LIN {X 0,Y 312.474,Z 713.562,A -85,B 0,C 180,E1 -15779.659,E2 -15779.659} C_VEL
LIN {X 0,Y 312.526,Z 713.531,A -85,B 0,C 180,E1 -15783.69,E2 -15783.69} C_VEL
LIN {X 0,Y 312.516,Z 713.544,A -85,B 0,C 180,E1 -15787.388,E2 -15787.388} C_VEL
LIN {X 0,Y 312.441,Z 713.564,A -85,B 0,C 180,E1 -15790.719,E2 -15790.719} C_VEL
LIN {X 0,Y 312.452,Z 713.564,A -85,B 0,C 180,E1 -15794.212,E2 -15794.212} C_VEL
LIN {X 0,Y 312.461,Z 713.565,A -85,B 0,C 180,E1 -15797.926,E2 -15797.926} C_VEL
LIN {X 0,Y 312.482,Z 713.562,A -85,B 0,C 180,E1 -15801.925,E2 -15801.925} C_VEL
LIN {X 0,Y 312.497,Z 713.558,A -85,B 0,C 180,E1 -15802.312,E2 -15802.312} C_VEL
LIN {X 0,Y 312.585,Z 714.3,A -85,B 0,C 180,E1 -15802.882,E2 -15802.882} C_VEL
LIN {X 0,Y 312.799,Z 716.737,A -85,B 0,C 180,E1 -15803.505,E2 -15803.505} C_VEL
LIN {X 0,Y 313.144,Z 721.496,A -85,B 0,C 180,E1 -15804.133,E2 -15804.133} C_VEL
LIN {X 0,Y 313.458,Z 727.496,A -85,B 0,C 180,E1 -15804.555,E2 -15804.555} C_VEL
LIN {X 0,Y 313.606,Z 731.828,A -85,B 0,C 180,E1 -15804.761,E2 -15804.761} C_VEL
LIN {X 0,Y 313.578,Z 740.657,A -85,B 0,C 180,E1 -15805.058,E2 -15805.058} C_VEL
LIN {X 0,Y 312.273,Z 790.691,A -85,B 0,C 180,E1 -15806.517,E2 -15806.517} C_VEL
LIN {X 0,Y 311.933,Z 803.373,A -85,B 0,C 180,E1 -15807.082,E2 -15807.082} C_VEL
LIN {X 0,Y 311.545,Z 814.797,A -85,B 0,C 180,E1 -15807.795,E2 -15807.795} C_VEL
LIN {X 0,Y 311.035,Z 823.817,A -85,B 0,C 180,E1 -15808.498,E2 -15808.498} C_VEL
LIN {X 0,Y 310.379,Z 833.968,A -85,B 0,C 180,E1 -15809.476,E2 -15809.476} C_VEL
LIN {X 0,Y 309.692,Z 843.6,A -85,B 0,C 180,E1 -15810.61,E2 -15810.61} C_VEL
LIN {X 0,Y 308.984,Z 852.175,A -85,B 0,C 180,E1 -15811.813,E2 -15811.813} C_VEL
LIN {X 0,Y 308.32,Z 860.705,A -85,B 0,C 180,E1 -15813.244,E2 -15813.244} C_VEL
LIN {X 0,Y 307.678,Z 867.783,A -85,B 0,C 180,E1 -15814.641,E2 -15814.641} C_VEL
LIN {X 0,Y 307.055,Z 874.035,A -85,B 0,C 180,E1 -15816.084,E2 -15816.084} C_VEL
LIN {X 0,Y 306.572,Z 880.144,A -85,B 0,C 180,E1 -15817.774,E2 -15817.774} C_VEL
LIN {X 0,Y 306.255,Z 884.439,A -85,B 0,C 180,E1 -15819.163,E2 -15819.163} C_VEL
LIN {X 0,Y 305.896,Z 889.538,A -85,B 0,C 180,E1 -15821.237,E2 -15821.237} C_VEL
LIN {X 0,Y 305.687,Z 893.372,A -85,B 0,C 180,E1 -15823.298,E2 -15823.298} C_VEL
LIN {X 0,Y 305.662,Z 896.085,A -85,B 0,C 180,E1 -15825.349,E2 -15825.349} C_VEL
LIN {X 0,Y 305.728,Z 897.387,A -85,B 0,C 180,E1 -15826.71,E2 -15826.71} C_VEL
LIN {X 0,Y 305.909,Z 898.143,A -85,B 0,C 180,E1 -15828.067,E2 -15828.067} C_VEL
LIN {X 0,Y 306.419,Z 898.401,A -85,B 0,C 180,E1 -15830.495,E2 -15830.495} C_VEL
LIN {X 0,Y 306.824,Z 897.718,A -85,B 0,C 180,E1 -15832.1,E2 -15832.1} C_VEL
LIN {X 0,Y 307.906,Z 895.323,A -85,B 0,C 180,E1 -15834.761,E2 -15834.761} C_VEL
LIN {X 0,Y 308.867,Z 892.287,A -85,B 0,C 180,E1 -15836.739,E2 -15836.739} C_VEL
LIN {X 0,Y 309.999,Z 888.123,A -85,B 0,C 180,E1 -15838.701,E2 -15838.701} C_VEL
LIN {X 0,Y 311.371,Z 882.681,A -85,B 0,C 180,E1 -15840.646,E2 -15840.646} C_VEL
LIN {X 0,Y 312.733,Z 877.075,A -85,B 0,C 180,E1 -15842.254,E2 -15842.254} C_VEL
LIN {X 0,Y 314.123,Z 870.334,A -85,B 0,C 180,E1 -15843.848,E2 -15843.848} C_VEL
LIN {X 0,Y 315.423,Z 864,A -85,B 0,C 180,E1 -15845.113,E2 -15845.113} C_VEL
LIN {X 0,Y 317.072,Z 854.397,A -85,B 0,C 180,E1 -15846.682,E2 -15846.682} C_VEL
LIN {X 0,Y 318.271,Z 846.362,A -85,B 0,C 180,E1 -15847.773,E2 -15847.773} C_VEL
LIN {X 0,Y 319.492,Z 836.672,A -85,B 0,C 180,E1 -15848.858,E2 -15848.858} C_VEL
LIN {X 0,Y 320.502,Z 826.458,A -85,B 0,C 180,E1 -15849.784,E2 -15849.784} C_VEL
LIN {X 0,Y 321.27,Z 816.948,A -85,B 0,C 180,E1 -15850.477,E2 -15850.477} C_VEL
LIN {X 0,Y 321.877,Z 806.465,A -85,B 0,C 180,E1 -15851.069,E2 -15851.069} C_VEL
LIN {X 0,Y 322.31,Z 791.848,A -85,B 0,C 180,E1 -15851.674,E2 -15851.674} C_VEL
LIN {X 0,Y 324.232,Z 756.607,A -85,B 0,C 180,E1 -15852.839,E2 -15852.839} C_VEL
LIN {X 0,Y 324.778,Z 747.442,A -85,B 0,C 180,E1 -15853.145,E2 -15853.145} C_VEL
LIN {X 0,Y 319.601,Z 737.334,A -85,B 0,C 180,E1 -15854.411,E2 -15854.411} C_VEL
LIN {X 0,Y 314.132,Z 727.873,A -85,B 0,C 180,E1 -15855.834,E2 -15855.834} C_VEL
LIN {X 0,Y 310.936,Z 723.294,A -85,B 0,C 180,E1 -15856.678,E2 -15856.678} C_VEL
LIN {X 0,Y 308.894,Z 719.974,A -85,B 0,C 180,E1 -15857.287,E2 -15857.287} C_VEL
LIN {X 0,Y 306.255,Z 716.727,A -85,B 0,C 180,E1 -15858.04,E2 -15858.04} C_VEL
LIN {X 0,Y 305.63,Z 714.906,A -85,B 0,C 180,E1 -15858.397,E2 -15858.397} C_VEL
LIN {X 0,Y 305.556,Z 714.458,A -85,B 0,C 180,E1 -15858.784,E2 -15858.784} C_VEL
LIN {X 0,Y 305.494,Z 714.431,A -85,B 0,C 180,E1 -15863.039,E2 -15863.039} C_VEL
LIN {X 0,Y 305.485,Z 714.434,A -85,B 0,C 180,E1 -15866.199,E2 -15866.199} C_VEL
LIN {X 0,Y 305.47,Z 714.433,A -85,B 0,C 180,E1 -15869.038,E2 -15869.038} C_VEL
LIN {X 0,Y 305.444,Z 714.437,A -85,B 0,C 180,E1 -15871.952,E2 -15871.952} C_VEL
LIN {X 0,Y 305.469,Z 714.433,A -85,B 0,C 180,E1 -15875.112,E2 -15875.112} C_VEL
LIN {X 0,Y 305.474,Z 714.432,A -85,B 0,C 180,E1 -15878.532,E2 -15878.532} C_VEL
LIN {X 0,Y 305.462,Z 714.434,A -85,B 0,C 180,E1 -15882.585,E2 -15882.585} C_VEL
LIN {X 0,Y 305.432,Z 714.44,A -85,B 0,C 180,E1 -15886.344,E2 -15886.344} C_VEL
LIN {X 0,Y 305.465,Z 714.437,A -85,B 0,C 180,E1 -15889.891,E2 -15889.891} C_VEL
LIN {X 0,Y 305.548,Z 714.64,A -85,B 0,C 180,E1 -15891.024,E2 -15891.024} C_VEL
LIN {X 0,Y 308.834,Z 727.96,A -85,B 0,C 180,E1 -15894.5,E2 -15894.5} C_VEL
LIN {X 0,Y 312.064,Z 742.523,A -85,B 0,C 180,E1 -15898.044,E2 -15898.044} C_VEL
LIN {X 0,Y 312.777,Z 746.093,A -85,B 0,C 180,E1 -15898.88,E2 -15898.88} C_VEL
LIN {X 0,Y 312.679,Z 749.371,A -85,B 0,C 180,E1 -15899.479,E2 -15899.479} C_VEL
LIN {X 0,Y 316.155,Z 773.114,A -85,B 0,C 180,E1 -15901.211,E2 -15901.211} C_VEL
LIN {X 0,Y 318.854,Z 797.479,A -85,B 0,C 180,E1 -15902.693,E2 -15902.693} C_VEL
LIN {X 0,Y 319.866,Z 811.457,A -85,B 0,C 180,E1 -15903.412,E2 -15903.412} C_VEL
LIN {X 0,Y 320.681,Z 834.523,A -85,B 0,C 180,E1 -15904.458,E2 -15904.458} C_VEL
LIN {X 0,Y 318.329,Z 876.074,A -85,B 0,C 180,E1 -15905.805,E2 -15905.805} C_VEL
LIN {X 0,Y 317.232,Z 887.509,A -85,B 0,C 180,E1 -15906.323,E2 -15906.323} C_VEL
LIN {X 0,Y 315.932,Z 898.532,A -85,B 0,C 180,E1 -15907.001,E2 -15907.001} C_VEL
LIN {X 0,Y 314.124,Z 911.078,A -85,B 0,C 180,E1 -15907.989,E2 -15907.989} C_VEL
LIN {X 0,Y 312.112,Z 923.208,A -85,B 0,C 180,E1 -15909.226,E2 -15909.226} C_VEL
LIN {X 0,Y 310.105,Z 934.166,A -85,B 0,C 180,E1 -15910.641,E2 -15910.641} C_VEL
LIN {X 0,Y 308.519,Z 943.318,A -85,B 0,C 180,E1 -15912.088,E2 -15912.088} C_VEL
LIN {X 0,Y 307.446,Z 950.333,A -85,B 0,C 180,E1 -15913.395,E2 -15913.395} C_VEL
LIN {X 0,Y 306.228,Z 957.721,A -85,B 0,C 180,E1 -15915.001,E2 -15915.001} C_VEL
LIN {X 0,Y 305.272,Z 965.314,A -85,B 0,C 180,E1 -15917.027,E2 -15917.027} C_VEL
LIN {X 0,Y 304.626,Z 972.881,A -85,B 0,C 180,E1 -15919.362,E2 -15919.362} C_VEL
LIN {X 0,Y 304.487,Z 978.046,A -85,B 0,C 180,E1 -15921.369,E2 -15921.369} C_VEL
LIN {X 0,Y 304.547,Z 982.046,A -85,B 0,C 180,E1 -15923.372,E2 -15923.372} C_VEL
LIN {X 0,Y 304.686,Z 984.103,A -85,B 0,C 180,E1 -15924.704,E2 -15924.704} C_VEL
LIN {X 0,Y 304.883,Z 985.727,A -85,B 0,C 180,E1 -15926.033,E2 -15926.033} C_VEL
LIN {X 0,Y 304.952,Z 986.88,A -85,B 0,C 180,E1 -15927.356,E2 -15927.356} C_VEL
LIN {X 0,Y 305.065,Z 987.581,A -85,B 0,C 180,E1 -15928.678,E2 -15928.678} C_VEL
LIN {X 0,Y 305.169,Z 987.868,A -85,B 0,C 180,E1 -15929.998,E2 -15929.998} C_VEL
LIN {X 0,Y 305.046,Z 987.713,A -85,B 0,C 180,E1 -15931.318,E2 -15931.318} C_VEL
LIN {X 0,Y 304.924,Z 987.132,A -85,B 0,C 180,E1 -15932.64,E2 -15932.64} C_VEL
LIN {X 0,Y 304.873,Z 986.11,A -85,B 0,C 180,E1 -15933.964,E2 -15933.964} C_VEL
LIN {X 0,Y 304.544,Z 982.776,A -85,B 0,C 180,E1 -15936.624,E2 -15936.624} C_VEL
LIN {X 0,Y 304.4,Z 979.067,A -85,B 0,C 180,E1 -15938.629,E2 -15938.629} C_VEL
LIN {X 0,Y 304.57,Z 974.278,A -85,B 0,C 180,E1 -15940.636,E2 -15940.636} C_VEL
LIN {X 0,Y 305.237,Z 967.143,A -85,B 0,C 180,E1 -15942.971,E2 -15942.971} C_VEL
LIN {X 0,Y 306.243,Z 959.332,A -85,B 0,C 180,E1 -15944.992,E2 -15944.992} C_VEL
LIN {X 0,Y 307.609,Z 950.031,A -85,B 0,C 180,E1 -15946.934,E2 -15946.934} C_VEL
LIN {X 0,Y 309.193,Z 940.33,A -85,B 0,C 180,E1 -15948.553,E2 -15948.553} C_VEL
LIN {X 0,Y 310.906,Z 929.646,A -85,B 0,C 180,E1 -15949.99,E2 -15949.99} C_VEL
LIN {X 0,Y 312.682,Z 917.833,A -85,B 0,C 180,E1 -15951.247,E2 -15951.247} C_VEL
LIN {X 0,Y 314.307,Z 905.31,A -85,B 0,C 180,E1 -15952.253,E2 -15952.253} C_VEL
LIN {X 0,Y 315.703,Z 892.229,A -85,B 0,C 180,E1 -15953.012,E2 -15953.012} C_VEL
LIN {X 0,Y 316.491,Z 879.543,A -85,B 0,C 180,E1 -15953.514,E2 -15953.514} C_VEL
LIN {X 0,Y 317.678,Z 830.97,A -85,B 0,C 180,E1 -15954.672,E2 -15954.672} C_VEL
LIN {X 0,Y 314.724,Z 799.143,A -85,B 0,C 180,E1 -15955.761,E2 -15955.761} C_VEL
LIN {X 0,Y 311.458,Z 773.975,A -85,B 0,C 180,E1 -15956.747,E2 -15956.747} C_VEL
LIN {X 0,Y 310.704,Z 768.362,A -85,B 0,C 180,E1 -15957.031,E2 -15957.031} C_VEL
LIN {X 0,Y 313.403,Z 749.284,A -85,B 0,C 180,E1 -15961.046,E2 -15961.046} C_VEL
LIN {X 0,Y 313.001,Z 745.438,A -85,B 0,C 180,E1 -15961.962,E2 -15961.962} C_VEL
LIN {X 0,Y 310.448,Z 733.482,A -85,B 0,C 180,E1 -15965.026,E2 -15965.026} C_VEL
LIN {X 0,Y 307.708,Z 722.464,A -85,B 0,C 180,E1 -15968.071,E2 -15968.071} C_VEL
LIN {X 0,Y 305.475,Z 714.541,A -85,B 0,C 180,E1 -15970.484,E2 -15970.484} C_VEL
LIN {X 0,Y 305.435,Z 714.433,A -85,B 0,C 180,E1 -15973.65,E2 -15973.65} C_VEL
LIN {X 0,Y 305.469,Z 714.432,A -85,B 0,C 180,E1 -15977.408,E2 -15977.408} C_VEL
LIN {X 0,Y 305.486,Z 714.43,A -85,B 0,C 180,E1 -15981.599,E2 -15981.599} C_VEL
LIN {X 0,Y 305.453,Z 714.418,A -85,B 0,C 180,E1 -15984.886,E2 -15984.886} C_VEL
LIN {X 0,Y 305.442,Z 714.435,A -85,B 0,C 180,E1 -15988.354,E2 -15988.354} C_VEL
LIN {X 0,Y 305.51,Z 714.428,A -85,B 0,C 180,E1 -15991.113,E2 -15991.113} C_VEL
LIN {X 0,Y 305.561,Z 714.42,A -85,B 0,C 180,E1 -15994.087,E2 -15994.087} C_VEL
LIN {X 0,Y 305.489,Z 714.424,A -85,B 0,C 180,E1 -15998.402,E2 -15998.402} C_VEL
LIN {X 0,Y 305.579,Z 714.421,A -85,B 0,C 180,E1 -16001.217,E2 -16001.217} C_VEL
LIN {X 0,Y 305.638,Z 714.414,A -85,B 0,C 180,E1 -16005.349,E2 -16005.349} C_VEL
LIN {X 0,Y 305.624,Z 714.415,A -85,B 0,C 180,E1 -16009.399,E2 -16009.399} C_VEL
LIN {X 0,Y 305.784,Z 714.387,A -85,B 0,C 180,E1 -16012.074,E2 -16012.074} C_VEL
LIN {X 0,Y 305.676,Z 714.402,A -85,B 0,C 180,E1 -16014.723,E2 -16014.723} C_VEL
LIN {X 0,Y 305.946,Z 714.372,A -85,B 0,C 180,E1 -16018.684,E2 -16018.684} C_VEL
LIN {X 0,Y 305.945,Z 714.371,A -85,B 0,C 180,E1 -16021.317,E2 -16021.317} C_VEL
LIN {X 0,Y 305.84,Z 714.39,A -85,B 0,C 180,E1 -16026.598,E2 -16026.598} C_VEL
LIN {X 0,Y 305.724,Z 714.397,A -85,B 0,C 180,E1 -16029.26,E2 -16029.26} C_VEL
LIN {X 0,Y 305.578,Z 714.418,A -85,B 0,C 180,E1 -16033.297,E2 -16033.297} C_VEL
LIN {X 0,Y 305.583,Z 714.412,A -85,B 0,C 180,E1 -16036.021,E2 -16036.021} C_VEL
LIN {X 0,Y 305.549,Z 714.42,A -85,B 0,C 180,E1 -16039.437,E2 -16039.437} C_VEL
LIN {X 0,Y 305.476,Z 714.414,A -85,B 0,C 180,E1 -16043.041,E2 -16043.041} C_VEL
LIN {X 0,Y 305.543,Z 714.428,A -85,B 0,C 180,E1 -16046.23,E2 -16046.23} C_VEL
LIN {X 0,Y 305.478,Z 714.419,A -85,B 0,C 180,E1 -16049.049,E2 -16049.049} C_VEL
LIN {X 0,Y 305.433,Z 714.431,A -85,B 0,C 180,E1 -16051.954,E2 -16051.954} C_VEL
LIN {X 0,Y 305.454,Z 714.432,A -85,B 0,C 180,E1 -16055.115,E2 -16055.115} C_VEL
LIN {X 0,Y 305.527,Z 714.61,A -85,B 0,C 180,E1 -16057.872,E2 -16057.872} C_VEL
LIN {X 0,Y 305.73,Z 715.512,A -85,B 0,C 180,E1 -16058.103,E2 -16058.103} C_VEL
LIN {X 0,Y 315.424,Z 734.481,A -85,B 0,C 180,E1 -16059.68,E2 -16059.68} C_VEL
LIN {X 0,Y 319.798,Z 744.244,A -85,B 0,C 180,E1 -16060.363,E2 -16060.363} C_VEL
LIN {X 0,Y 318.757,Z 791.246,A -85,B 0,C 180,E1 -16061.487,E2 -16061.487} C_VEL
LIN {X 0,Y 318.629,Z 805.311,A -85,B 0,C 180,E1 -16061.953,E2 -16061.953} C_VEL
LIN {X 0,Y 318.217,Z 817.903,A -85,B 0,C 180,E1 -16062.635,E2 -16062.635} C_VEL
LIN {X 0,Y 317.446,Z 829.918,A -85,B 0,C 180,E1 -16063.529,E2 -16063.529} C_VEL
LIN {X 0,Y 316.275,Z 841.723,A -85,B 0,C 180,E1 -16064.68,E2 -16064.68} C_VEL
LIN {X 0,Y 315.059,Z 851.984,A -85,B 0,C 180,E1 -16065.965,E2 -16065.965} C_VEL
LIN {X 0,Y 313.601,Z 862.112,A -85,B 0,C 180,E1 -16067.539,E2 -16067.539} C_VEL
LIN {X 0,Y 312.162,Z 870.912,A -85,B 0,C 180,E1 -16069.242,E2 -16069.242} C_VEL
LIN {X 0,Y 310.744,Z 878.712,A -85,B 0,C 180,E1 -16071.129,E2 -16071.129} C_VEL
LIN {X 0,Y 309.477,Z 885.377,A -85,B 0,C 180,E1 -16073.155,E2 -16073.155} C_VEL
LIN {X 0,Y 308.311,Z 890.805,A -85,B 0,C 180,E1 -16075.261,E2 -16075.261} C_VEL
LIN {X 0,Y 307.625,Z 893.802,A -85,B 0,C 180,E1 -16076.752,E2 -16076.752} C_VEL
LIN {X 0,Y 307.12,Z 896.217,A -85,B 0,C 180,E1 -16078.245,E2 -16078.245} C_VEL
LIN {X 0,Y 306.516,Z 898.862,A -85,B 0,C 180,E1 -16080.61,E2 -16080.61} C_VEL
LIN {X 0,Y 306.113,Z 900.115,A -85,B 0,C 180,E1 -16082.668,E2 -16082.668} C_VEL
LIN {X 0,Y 305.972,Z 900.399,A -85,B 0,C 180,E1 -16084.127,E2 -16084.127} C_VEL
LIN {X 0,Y 305.894,Z 900.247,A -85,B 0,C 180,E1 -16085.574,E2 -16085.574} C_VEL
LIN {X 0,Y 305.928,Z 899.592,A -85,B 0,C 180,E1 -16087.014,E2 -16087.014} C_VEL
LIN {X 0,Y 306.068,Z 898.48,A -85,B 0,C 180,E1 -16088.447,E2 -16088.447} C_VEL
LIN {X 0,Y 306.371,Z 896.552,A -85,B 0,C 180,E1 -16090.141,E2 -16090.141} C_VEL
LIN {X 0,Y 307.026,Z 892.313,A -85,B 0,C 180,E1 -16092.69,E2 -16092.69} C_VEL
LIN {X 0,Y 307.806,Z 887.5,A -85,B 0,C 180,E1 -16094.779,E2 -16094.779} C_VEL
LIN {X 0,Y 308.726,Z 881.356,A -85,B 0,C 180,E1 -16096.844,E2 -16096.844} C_VEL
LIN {X 0,Y 309.865,Z 873.672,A -85,B 0,C 180,E1 -16098.887,E2 -16098.887} C_VEL
LIN {X 0,Y 310.965,Z 865.834,A -85,B 0,C 180,E1 -16100.571,E2 -16100.571} C_VEL
LIN {X 0,Y 312.203,Z 856.299,A -85,B 0,C 180,E1 -16102.24,E2 -16102.24} C_VEL
LIN {X 0,Y 313.404,Z 845.67,A -85,B 0,C 180,E1 -16103.726,E2 -16103.726} C_VEL
LIN {X 0,Y 314.523,Z 833.894,A -85,B 0,C 180,E1 -16105.035,E2 -16105.035} C_VEL
LIN {X 0,Y 315.393,Z 821.458,A -85,B 0,C 180,E1 -16106.089,E2 -16106.089} C_VEL
LIN {X 0,Y 315.943,Z 808.598,A -85,B 0,C 180,E1 -16106.894,E2 -16106.894} C_VEL
LIN {X 0,Y 316.171,Z 796.443,A -85,B 0,C 180,E1 -16107.414,E2 -16107.414} C_VEL
LIN {X 0,Y 316.968,Z 746.283,A -85,B 0,C 180,E1 -16108.625,E2 -16108.625} C_VEL
LIN {X 0,Y 317.049,Z 741.291,A -85,B 0,C 180,E1 -16108.743,E2 -16108.743} C_VEL
LIN {X 0,Y 309.365,Z 722.642,A -85,B 0,C 180,E1 -16109.816,E2 -16109.816} C_VEL
LIN {X 0,Y 306.062,Z 715.169,A -85,B 0,C 180,E1 -16110.331,E2 -16110.331} C_VEL
LIN {X 0,Y 305.923,Z 714.461,A -85,B 0,C 180,E1 -16110.578,E2 -16110.578} C_VEL
LIN {X 0,Y 305.85,Z 714.387,A -85,B 0,C 180,E1 -16112.636,E2 -16112.636} C_VEL
LIN {X 0,Y 305.788,Z 714.391,A -85,B 0,C 180,E1 -16116.601,E2 -16116.601} C_VEL
LIN {X 0,Y 305.698,Z 714.406,A -85,B 0,C 180,E1 -16119.263,E2 -16119.263} C_VEL
LIN {X 0,Y 305.589,Z 714.417,A -85,B 0,C 180,E1 -16123.298,E2 -16123.298} C_VEL
LIN {X 0,Y 305.554,Z 714.418,A -85,B 0,C 180,E1 -16126.024,E2 -16126.024} C_VEL
LIN {X 0,Y 305.485,Z 714.414,A -85,B 0,C 180,E1 -16130.189,E2 -16130.189} C_VEL
LIN {X 0,Y 305.461,Z 714.431,A -85,B 0,C 180,E1 -16134.467,E2 -16134.467} C_VEL
LIN {X 0,Y 305.447,Z 714.418,A -85,B 0,C 180,E1 -16137.401,E2 -16137.401} C_VEL
LIN {X 0,Y 305.421,Z 714.439,A -85,B 0,C 180,E1 -16140.416,E2 -16140.416} C_VEL
LIN {X 0,Y 305.471,Z 714.406,A -85,B 0,C 180,E1 -16144.079,E2 -16144.079} C_VEL
LIN {X 0,Y 305.458,Z 714.418,A -85,B 0,C 180,E1 -16146.744,E2 -16146.744} C_VEL
LIN {X 0,Y 305.412,Z 714.439,A -85,B 0,C 180,E1 -16150.59,E2 -16150.59} C_VEL
LIN {X 0,Y 305.402,Z 714.442,A -85,B 0,C 180,E1 -16154.489,E2 -16154.489} C_VEL
LIN {X 0,Y 305.418,Z 714.441,A -85,B 0,C 180,E1 -16158.139,E2 -16158.139} C_VEL
LIN {X 0,Y 305.444,Z 714.434,A -85,B 0,C 180,E1 -16162.318,E2 -16162.318} C_VEL
LIN {X 0,Y 305.515,Z 714.584,A -85,B 0,C 180,E1 -16163.626,E2 -16163.626} C_VEL
LIN {X 0,Y 305.74,Z 715.565,A -85,B 0,C 180,E1 -16163.847,E2 -16163.847} C_VEL
LIN {X 0,Y 313.568,Z 737.666,A -85,B 0,C 180,E1 -16164.965,E2 -16164.965} C_VEL
LIN {X 0,Y 313.578,Z 740.657,A -85,B 0,C 180,E1 -16165.058,E2 -16165.058} C_VEL
LIN {X 0,Y 312.734,Z 746.454,A -85,B 0,C 180,E1 -16165.195,E2 -16165.195} C_VEL
LIN {X 0,Y 306.578,Z 765.245,A -85,B 0,C 180,E1 -16165.463,E2 -16165.463} C_VEL
LIN {X 0,Y 305.777,Z 771.044,A -85,B 0,C 180,E1 -16165.605,E2 -16165.605} C_VEL
LIN {X 0,Y 305.326,Z 794.538,A -85,B 0,C 180,E1 -16166.36,E2 -16166.36} C_VEL
LIN {X 0,Y 305.001,Z 805.646,A -85,B 0,C 180,E1 -16166.894,E2 -16166.894} C_VEL
LIN {X 0,Y 304.593,Z 815.918,A -85,B 0,C 180,E1 -16167.557,E2 -16167.557} C_VEL
LIN {X 0,Y 304.024,Z 825.634,A -85,B 0,C 180,E1 -16168.343,E2 -16168.343} C_VEL
LIN {X 0,Y 303.35,Z 835.762,A -85,B 0,C 180,E1 -16169.356,E2 -16169.356} C_VEL
LIN {X 0,Y 302.706,Z 844.701,A -85,B 0,C 180,E1 -16170.438,E2 -16170.438} C_VEL
LIN {X 0,Y 301.987,Z 853.411,A -85,B 0,C 180,E1 -16171.694,E2 -16171.694} C_VEL
LIN {X 0,Y 301.387,Z 860.846,A -85,B 0,C 180,E1 -16172.953,E2 -16172.953} C_VEL
LIN {X 0,Y 300.712,Z 868.066,A -85,B 0,C 180,E1 -16174.382,E2 -16174.382} C_VEL
LIN {X 0,Y 300.009,Z 875.015,A -85,B 0,C 180,E1 -16176.014,E2 -16176.014} C_VEL
LIN {X 0,Y 299.496,Z 881.754,A -85,B 0,C 180,E1 -16177.947,E2 -16177.947} C_VEL
LIN {X 0,Y 299.161,Z 885.968,A -85,B 0,C 180,E1 -16179.366,E2 -16179.366} C_VEL
LIN {X 0,Y 298.805,Z 890.961,A -85,B 0,C 180,E1 -16181.486,E2 -16181.486} C_VEL
LIN {X 0,Y 298.635,Z 894.723,A -85,B 0,C 180,E1 -16183.596,E2 -16183.596} C_VEL
LIN {X 0,Y 298.642,Z 896.698,A -85,B 0,C 180,E1 -16184.997,E2 -16184.997} C_VEL
LIN {X 0,Y 298.85,Z 899.05,A -85,B 0,C 180,E1 -16187.781,E2 -16187.781} C_VEL
LIN {X 0,Y 299.107,Z 899.551,A -85,B 0,C 180,E1 -16189.165,E2 -16189.165} C_VEL
LIN {X 0,Y 299.431,Z 899.584,A -85,B 0,C 180,E1 -16190.543,E2 -16190.543} C_VEL
LIN {X 0,Y 300.297,Z 898.379,A -85,B 0,C 180,E1 -16193.28,E2 -16193.28} C_VEL
LIN {X 0,Y 300.883,Z 897.05,A -85,B 0,C 180,E1 -16194.639,E2 -16194.639} C_VEL
LIN {X 0,Y 302.263,Z 893.151,A -85,B 0,C 180,E1 -16197.334,E2 -16197.334} C_VEL
LIN {X 0,Y 303.496,Z 888.881,A -85,B 0,C 180,E1 -16199.336,E2 -16199.336} C_VEL
LIN {X 0,Y 304.999,Z 883.346,A -85,B 0,C 180,E1 -16201.32,E2 -16201.32} C_VEL
LIN {X 0,Y 306.479,Z 877.671,A -85,B 0,C 180,E1 -16202.957,E2 -16202.957} C_VEL
LIN {X 0,Y 307.681,Z 872.391,A -85,B 0,C 180,E1 -16204.257,E2 -16204.257} C_VEL
LIN {X 0,Y 309.386,Z 864.367,A -85,B 0,C 180,E1 -16205.867,E2 -16205.867} C_VEL
LIN {X 0,Y 310.799,Z 856.743,A -85,B 0,C 180,E1 -16207.144,E2 -16207.144} C_VEL
LIN {X 0,Y 312.264,Z 847.644,A -85,B 0,C 180,E1 -16208.412,E2 -16208.412} C_VEL
LIN {X 0,Y 313.528,Z 838.356,A -85,B 0,C 180,E1 -16209.487,E2 -16209.487} C_VEL
LIN {X 0,Y 314.524,Z 829.875,A -85,B 0,C 180,E1 -16210.297,E2 -16210.297} C_VEL
LIN {X 0,Y 315.362,Z 819.879,A -85,B 0,C 180,E1 -16211.082,E2 -16211.082} C_VEL
LIN {X 0,Y 316.103,Z 808.632,A -85,B 0,C 180,E1 -16211.746,E2 -16211.746} C_VEL
LIN {X 0,Y 316.552,Z 795.014,A -85,B 0,C 180,E1 -16212.339,E2 -16212.339} C_VEL
LIN {X 0,Y 318.225,Z 765.799,A -85,B 0,C 180,E1 -16213.349,E2 -16213.349} C_VEL
LIN {X 0,Y 319.277,Z 750.021,A -85,B 0,C 180,E1 -16213.886,E2 -16213.886} C_VEL
LIN {X 0,Y 313.25,Z 738.49,A -85,B 0,C 180,E1 -16215.462,E2 -16215.462} C_VEL
LIN {X 0,Y 308.903,Z 731.443,A -85,B 0,C 180,E1 -16216.657,E2 -16216.657} C_VEL
LIN {X 0,Y 306.662,Z 728.003,A -85,B 0,C 180,E1 -16217.323,E2 -16217.323} C_VEL
LIN {X 0,Y 304.411,Z 724.587,A -85,B 0,C 180,E1 -16218.007,E2 -16218.007} C_VEL
LIN {X 0,Y 302.286,Z 721.473,A -85,B 0,C 180,E1 -16218.691,E2 -16218.691} C_VEL
LIN {X 0,Y 301.699,Z 720.414,A -85,B 0,C 180,E1 -16218.899,E2 -16218.899} C_VEL
LIN {X 0,Y 299.389,Z 717.967,A -85,B 0,C 180,E1 -16219.633,E2 -16219.633} C_VEL
LIN {X 0,Y 298.573,Z 715.892,A -85,B 0,C 180,E1 -16220.072,E2 -16220.072} C_VEL
LIN {X 0,Y 298.441,Z 715.323,A -85,B 0,C 180,E1 -16220.685,E2 -16220.685} C_VEL
LIN {X 0,Y 298.457,Z 715.306,A -85,B 0,C 180,E1 -16225.078,E2 -16225.078} C_VEL
LIN {X 0,Y 298.418,Z 715.314,A -85,B 0,C 180,E1 -16229.377,E2 -16229.377} C_VEL
LIN {X 0,Y 298.4,Z 715.313,A -85,B 0,C 180,E1 -16232.8,E2 -16232.8} C_VEL
LIN {X 0,Y 298.458,Z 715.305,A -85,B 0,C 180,E1 -16236.808,E2 -16236.808} C_VEL
LIN {X 0,Y 298.416,Z 715.312,A -85,B 0,C 180,E1 -16239.485,E2 -16239.485} C_VEL
LIN {X 0,Y 298.405,Z 715.312,A -85,B 0,C 180,E1 -16243.102,E2 -16243.102} C_VEL
LIN {X 0,Y 298.409,Z 715.312,A -85,B 0,C 180,E1 -16246.92,E2 -16246.92} C_VEL
LIN {X 0,Y 298.465,Z 715.403,A -85,B 0,C 180,E1 -16250.411,E2 -16250.411} C_VEL
LIN {X 0,Y 299.21,Z 718.35,A -85,B 0,C 180,E1 -16251.304,E2 -16251.304} C_VEL
LIN {X 0,Y 302.683,Z 732.696,A -85,B 0,C 180,E1 -16255.07,E2 -16255.07} C_VEL
LIN {X 0,Y 304.493,Z 740.8,A -85,B 0,C 180,E1 -16257.065,E2 -16257.065} C_VEL
LIN {X 0,Y 306.204,Z 747.221,A -85,B 0,C 180,E1 -16258.135,E2 -16258.135} C_VEL
LIN {X 0,Y 307.688,Z 752.126,A -85,B 0,C 180,E1 -16258.693,E2 -16258.693} C_VEL
LIN {X 0,Y 310.905,Z 775.277,A -85,B 0,C 180,E1 -16260.438,E2 -16260.438} C_VEL
LIN {X 0,Y 313.325,Z 798.973,A -85,B 0,C 180,E1 -16261.934,E2 -16261.934} C_VEL
LIN {X 0,Y 314.23,Z 813.346,A -85,B 0,C 180,E1 -16262.706,E2 -16262.706} C_VEL
LIN {X 0,Y 314.908,Z 835.446,A -85,B 0,C 180,E1 -16263.729,E2 -16263.729} C_VEL
LIN {X 0,Y 312.474,Z 874.755,A -85,B 0,C 180,E1 -16265.055,E2 -16265.055} C_VEL
LIN {X 0,Y 311.232,Z 886.765,A -85,B 0,C 180,E1 -16265.616,E2 -16265.616} C_VEL
LIN {X 0,Y 309.486,Z 900.437,A -85,B 0,C 180,E1 -16266.494,E2 -16266.494} C_VEL
LIN {X 0,Y 307.327,Z 913.607,A -85,B 0,C 180,E1 -16267.653,E2 -16267.653} C_VEL
LIN {X 0,Y 305.506,Z 923.608,A -85,B 0,C 180,E1 -16268.755,E2 -16268.755} C_VEL
LIN {X 0,Y 303.676,Z 933.179,A -85,B 0,C 180,E1 -16270.038,E2 -16270.038} C_VEL
LIN {X 0,Y 302.14,Z 941.379,A -85,B 0,C 180,E1 -16271.345,E2 -16271.345} C_VEL
LIN {X 0,Y 300.816,Z 948.49,A -85,B 0,C 180,E1 -16272.668,E2 -16272.668} C_VEL
LIN {X 0,Y 299.392,Z 956.315,A -85,B 0,C 180,E1 -16274.411,E2 -16274.411} C_VEL
LIN {X 0,Y 298.416,Z 963.57,A -85,B 0,C 180,E1 -16276.376,E2 -16276.376} C_VEL
LIN {X 0,Y 297.742,Z 969.781,A -85,B 0,C 180,E1 -16278.424,E2 -16278.424} C_VEL
LIN {X 0,Y 297.451,Z 975.316,A -85,B 0,C 180,E1 -16280.478,E2 -16280.478} C_VEL
LIN {X 0,Y 297.453,Z 980.432,A -85,B 0,C 180,E1 -16282.907,E2 -16282.907} C_VEL
LIN {X 0,Y 297.617,Z 983.026,A -85,B 0,C 180,E1 -16284.578,E2 -16284.578} C_VEL
LIN {X 0,Y 297.836,Z 984.665,A -85,B 0,C 180,E1 -16285.939,E2 -16285.939} C_VEL
LIN {X 0,Y 297.908,Z 985.84,A -85,B 0,C 180,E1 -16287.294,E2 -16287.294} C_VEL
LIN {X 0,Y 298.028,Z 986.554,A -85,B 0,C 180,E1 -16288.647,E2 -16288.647} C_VEL
LIN {X 0,Y 298.139,Z 986.852,A -85,B 0,C 180,E1 -16289.998,E2 -16289.998} C_VEL
LIN {X 0,Y 298.007,Z 986.704,A -85,B 0,C 180,E1 -16291.349,E2 -16291.349} C_VEL
LIN {X 0,Y 297.877,Z 986.139,A -85,B 0,C 180,E1 -16292.703,E2 -16292.703} C_VEL
LIN {X 0,Y 297.804,Z 985.124,A -85,B 0,C 180,E1 -16294.058,E2 -16294.058} C_VEL
LIN {X 0,Y 297.567,Z 983.666,A -85,B 0,C 180,E1 -16295.419,E2 -16295.419} C_VEL
LIN {X 0,Y 297.428,Z 981.381,A -85,B 0,C 180,E1 -16297.055,E2 -16297.055} C_VEL
LIN {X 0,Y 297.344,Z 976.633,A -85,B 0,C 180,E1 -16299.521,E2 -16299.521} C_VEL
LIN {X 0,Y 297.679,Z 971.482,A -85,B 0,C 180,E1 -16301.575,E2 -16301.575} C_VEL
LIN {X 0,Y 298.347,Z 965.075,A -85,B 0,C 180,E1 -16303.623,E2 -16303.623} C_VEL
LIN {X 0,Y 299.226,Z 958.883,A -85,B 0,C 180,E1 -16305.253,E2 -16305.253} C_VEL
LIN {X 0,Y 300.762,Z 949.241,A -85,B 0,C 180,E1 -16307.331,E2 -16307.331} C_VEL
LIN {X 0,Y 302.455,Z 939.616,A -85,B 0,C 180,E1 -16308.982,E2 -16308.982} C_VEL
LIN {X 0,Y 304.246,Z 929.001,A -85,B 0,C 180,E1 -16310.447,E2 -16310.447} C_VEL
LIN {X 0,Y 305.791,Z 918.876,A -85,B 0,C 180,E1 -16311.573,E2 -16311.573} C_VEL
LIN {X 0,Y 307.475,Z 907.101,A -85,B 0,C 180,E1 -16312.597,E2 -16312.597} C_VEL
LIN {X 0,Y 308.941,Z 894.403,A -85,B 0,C 180,E1 -16313.413,E2 -16313.413} C_VEL
LIN {X 0,Y 309.945,Z 881.094,A -85,B 0,C 180,E1 -16313.997,E2 -16313.997} C_VEL
LIN {X 0,Y 310.793,Z 855.297,A -85,B 0,C 180,E1 -16314.653,E2 -16314.653} C_VEL
LIN {X 0,Y 311.281,Z 831.143,A -85,B 0,C 180,E1 -16315.242,E2 -16315.242} C_VEL
LIN {X 0,Y 308.408,Z 799.908,A -85,B 0,C 180,E1 -16316.35,E2 -16316.35} C_VEL
LIN {X 0,Y 305.525,Z 777.341,A -85,B 0,C 180,E1 -16317.255,E2 -16317.255} C_VEL
LIN {X 0,Y 304.078,Z 767.429,A -85,B 0,C 180,E1 -16317.719,E2 -16317.719} C_VEL
LIN {X 0,Y 306.633,Z 750.18,A -85,B 0,C 180,E1 -16321.425,E2 -16321.425} C_VEL
LIN {X 0,Y 304.61,Z 739.442,A -85,B 0,C 180,E1 -16324.182,E2 -16324.182} C_VEL
LIN {X 0,Y 301.678,Z 727.061,A -85,B 0,C 180,E1 -16327.62,E2 -16327.62} C_VEL
LIN {X 0,Y 298.837,Z 717.039,A -85,B 0,C 180,E1 -16330.672,E2 -16330.672} C_VEL
LIN {X 0,Y 298.398,Z 715.405,A -85,B 0,C 180,E1 -16331.256,E2 -16331.256} C_VEL
LIN {X 0,Y 298.38,Z 715.315,A -85,B 0,C 180,E1 -16335.04,E2 -16335.04} C_VEL
LIN {X 0,Y 298.404,Z 715.31,A -85,B 0,C 180,E1 -16338.742,E2 -16338.742} C_VEL
LIN {X 0,Y 298.422,Z 715.313,A -85,B 0,C 180,E1 -16342.243,E2 -16342.243} C_VEL
LIN {X 0,Y 298.398,Z 715.301,A -85,B 0,C 180,E1 -16345.58,E2 -16345.58} C_VEL
LIN {X 0,Y 298.385,Z 715.313,A -85,B 0,C 180,E1 -16348.79,E2 -16348.79} C_VEL
LIN {X 0,Y 298.459,Z 715.303,A -85,B 0,C 180,E1 -16351.904,E2 -16351.904} C_VEL
LIN {X 0,Y 298.475,Z 715.3,A -85,B 0,C 180,E1 -16354.923,E2 -16354.923} C_VEL
LIN {X 0,Y 298.439,Z 715.303,A -85,B 0,C 180,E1 -16359.315,E2 -16359.315} C_VEL
LIN {X 0,Y 298.526,Z 715.29,A -85,B 0,C 180,E1 -16362.179,E2 -16362.179} C_VEL
LIN {X 0,Y 298.582,Z 715.291,A -85,B 0,C 180,E1 -16364.994,E2 -16364.994} C_VEL
LIN {X 0,Y 298.58,Z 715.292,A -85,B 0,C 180,E1 -16369.146,E2 -16369.146} C_VEL
LIN {X 0,Y 298.729,Z 715.264,A -85,B 0,C 180,E1 -16371.885,E2 -16371.885} C_VEL
LIN {X 0,Y 298.646,Z 715.279,A -85,B 0,C 180,E1 -16374.599,E2 -16374.599} C_VEL
LIN {X 0,Y 298.912,Z 715.248,A -85,B 0,C 180,E1 -16378.653,E2 -16378.653} C_VEL
LIN {X 0,Y 298.912,Z 715.247,A -85,B 0,C 180,E1 -16381.347,E2 -16381.347} C_VEL
LIN {X 0,Y 298.785,Z 715.268,A -85,B 0,C 180,E1 -16386.754,E2 -16386.754} C_VEL
LIN {X 0,Y 298.669,Z 715.277,A -85,B 0,C 180,E1 -16389.481,E2 -16389.481} C_VEL
LIN {X 0,Y 298.541,Z 715.297,A -85,B 0,C 180,E1 -16393.616,E2 -16393.616} C_VEL
LIN {X 0,Y 298.538,Z 715.291,A -85,B 0,C 180,E1 -16396.41,E2 -16396.41} C_VEL
LIN {X 0,Y 298.487,Z 715.3,A -85,B 0,C 180,E1 -16399.648,E2 -16399.648} C_VEL
LIN {X 0,Y 298.418,Z 715.291,A -85,B 0,C 180,E1 -16403.601,E2 -16403.601} C_VEL
LIN {X 0,Y 298.481,Z 715.308,A -85,B 0,C 180,E1 -16406.576,E2 -16406.576} C_VEL
LIN {X 0,Y 298.407,Z 715.305,A -85,B 0,C 180,E1 -16409.643,E2 -16409.643} C_VEL
LIN {X 0,Y 298.386,Z 715.305,A -85,B 0,C 180,E1 -16412.802,E2 -16412.802} C_VEL
LIN {X 0,Y 298.492,Z 715.476,A -85,B 0,C 180,E1 -16417.072,E2 -16417.072} C_VEL
LIN {X 0,Y 298.761,Z 716.615,A -85,B 0,C 180,E1 -16417.343,E2 -16417.343} C_VEL
LIN {X 0,Y 307.419,Z 733.091,A -85,B 0,C 180,E1 -16418.805,E2 -16418.805} C_VEL
LIN {X 0,Y 313.512,Z 746.196,A -85,B 0,C 180,E1 -16419.801,E2 -16419.801} C_VEL
LIN {X 0,Y 312.432,Z 792.282,A -85,B 0,C 180,E1 -16420.926,E2 -16420.926} C_VEL
LIN {X 0,Y 312.298,Z 805.781,A -85,B 0,C 180,E1 -16421.375,E2 -16421.375} C_VEL
LIN {X 0,Y 311.939,Z 817.079,A -85,B 0,C 180,E1 -16421.974,E2 -16421.974} C_VEL
LIN {X 0,Y 311.204,Z 828.851,A -85,B 0,C 180,E1 -16422.83,E2 -16422.83} C_VEL
LIN {X 0,Y 310.08,Z 840.427,A -85,B 0,C 180,E1 -16423.928,E2 -16423.928} C_VEL
LIN {X 0,Y 308.903,Z 850.544,A -85,B 0,C 180,E1 -16425.15,E2 -16425.15} C_VEL
LIN {X 0,Y 307.402,Z 860.839,A -85,B 0,C 180,E1 -16426.699,E2 -16426.699} C_VEL
LIN {X 0,Y 305.993,Z 869.13,A -85,B 0,C 180,E1 -16428.239,E2 -16428.239} C_VEL
LIN {X 0,Y 304.45,Z 877.518,A -85,B 0,C 180,E1 -16430.167,E2 -16430.167} C_VEL
LIN {X 0,Y 303.199,Z 883.949,A -85,B 0,C 180,E1 -16432.009,E2 -16432.009} C_VEL
LIN {X 0,Y 302.196,Z 888.572,A -85,B 0,C 180,E1 -16433.63,E2 -16433.63} C_VEL
LIN {X 0,Y 300.966,Z 893.743,A -85,B 0,C 180,E1 -16435.917,E2 -16435.917} C_VEL
LIN {X 0,Y 300.117,Z 897.475,A -85,B 0,C 180,E1 -16438.207,E2 -16438.207} C_VEL
LIN {X 0,Y 299.546,Z 899.9,A -85,B 0,C 180,E1 -16440.484,E2 -16440.484} C_VEL
LIN {X 0,Y 299.201,Z 900.872,A -85,B 0,C 180,E1 -16441.982,E2 -16441.982} C_VEL
LIN {X 0,Y 299.027,Z 901.379,A -85,B 0,C 180,E1 -16443.48,E2 -16443.48} C_VEL
LIN {X 0,Y 298.897,Z 901.366,A -85,B 0,C 180,E1 -16444.963,E2 -16444.963} C_VEL
LIN {X 0,Y 298.884,Z 900.884,A -85,B 0,C 180,E1 -16446.5,E2 -16446.5} C_VEL
LIN {X 0,Y 298.997,Z 899.99,A -85,B 0,C 180,E1 -16447.911,E2 -16447.911} C_VEL
LIN {X 0,Y 299.289,Z 897.936,A -85,B 0,C 180,E1 -16449.935,E2 -16449.935} C_VEL
LIN {X 0,Y 299.882,Z 894.355,A -85,B 0,C 180,E1 -16452.264,E2 -16452.264} C_VEL
LIN {X 0,Y 300.601,Z 889.848,A -85,B 0,C 180,E1 -16454.405,E2 -16454.405} C_VEL
LIN {X 0,Y 301.542,Z 884.065,A -85,B 0,C 180,E1 -16456.524,E2 -16456.524} C_VEL
LIN {X 0,Y 302.677,Z 876.837,A -85,B 0,C 180,E1 -16458.619,E2 -16458.619} C_VEL
LIN {X 0,Y 304.003,Z 867.749,A -85,B 0,C 180,E1 -16460.689,E2 -16460.689} C_VEL
LIN {X 0,Y 305.282,Z 858.472,A -85,B 0,C 180,E1 -16462.386,E2 -16462.386} C_VEL
LIN {X 0,Y 306.541,Z 848.084,A -85,B 0,C 180,E1 -16463.915,E2 -16463.915} C_VEL
LIN {X 0,Y 307.681,Z 836.632,A -85,B 0,C 180,E1 -16465.252,E2 -16465.252} C_VEL
LIN {X 0,Y 308.644,Z 824.793,A -85,B 0,C 180,E1 -16466.33,E2 -16466.33} C_VEL
LIN {X 0,Y 309.224,Z 812.126,A -85,B 0,C 180,E1 -16467.193,E2 -16467.193} C_VEL
LIN {X 0,Y 309.536,Z 798.303,A -85,B 0,C 180,E1 -16467.833,E2 -16467.833} C_VEL
LIN {X 0,Y 310.213,Z 754.752,A -85,B 0,C 180,E1 -16468.927,E2 -16468.927} C_VEL
LIN {X 0,Y 310.374,Z 742.878,A -85,B 0,C 180,E1 -16469.217,E2 -16469.217} C_VEL
LIN {X 0,Y 303.28,Z 725.574,A -85,B 0,C 180,E1 -16470.242,E2 -16470.242} C_VEL
LIN {X 0,Y 299.07,Z 716.201,A -85,B 0,C 180,E1 -16470.886,E2 -16470.886} C_VEL
LIN {X 0,Y 298.909,Z 715.32,A -85,B 0,C 180,E1 -16471.181,E2 -16471.181} C_VEL
LIN {X 0,Y 298.628,Z 715.289,A -85,B 0,C 180,E1 -16475.404,E2 -16475.404} C_VEL
LIN {X 0,Y 298.702,Z 715.274,A -85,B 0,C 180,E1 -16478.118,E2 -16478.118} C_VEL
LIN {X 0,Y 298.552,Z 715.295,A -85,B 0,C 180,E1 -16482.233,E2 -16482.233} C_VEL
LIN {X 0,Y 298.553,Z 715.284,A -85,B 0,C 180,E1 -16485.169,E2 -16485.169} C_VEL
LIN {X 0,Y 298.444,Z 715.292,A -85,B 0,C 180,E1 -16489.617,E2 -16489.617} C_VEL
LIN {X 0,Y 298.394,Z 715.314,A -85,B 0,C 180,E1 -16493.605,E2 -16493.605} C_VEL
LIN {X 0,Y 298.407,Z 715.291,A -85,B 0,C 180,E1 -16496.584,E2 -16496.584} C_VEL
LIN {X 0,Y 298.362,Z 715.32,A -85,B 0,C 180,E1 -16499.649,E2 -16499.649} C_VEL
LIN {X 0,Y 298.398,Z 715.3,A -85,B 0,C 180,E1 -16502.802,E2 -16502.802} C_VEL
LIN {X 0,Y 298.41,Z 715.288,A -85,B 0,C 180,E1 -16506.073,E2 -16506.073} C_VEL
LIN {X 0,Y 298.38,Z 715.319,A -85,B 0,C 180,E1 -16509.493,E2 -16509.493} C_VEL
LIN {X 0,Y 298.373,Z 715.318,A -85,B 0,C 180,E1 -16513.097,E2 -16513.097} C_VEL
LIN {X 0,Y 298.376,Z 715.317,A -85,B 0,C 180,E1 -16516.915,E2 -16516.915} C_VEL
LIN {X 0,Y 298.392,Z 715.317,A -85,B 0,C 180,E1 -16521.012,E2 -16521.012} C_VEL
LIN {X 0,Y 298.525,Z 715.594,A -85,B 0,C 180,E1 -16523.312,E2 -16523.312} C_VEL
LIN {X 0,Y 298.694,Z 716.39,A -85,B 0,C 180,E1 -16523.469,E2 -16523.469} C_VEL
LIN {X 0,Y 306.741,Z 739.202,A -85,B 0,C 180,E1 -16524.663,E2 -16524.663} C_VEL
LIN {X 0,Y 305.777,Z 771.044,A -85,B 0,C 180,E1 -16525.605,E2 -16525.605} C_VEL
LIN {X 0,Y 305.013,Z 776.842,A -85,B 0,C 180,E1 -16525.744,E2 -16525.744} C_VEL
LIN {X 0,Y 299.166,Z 795.643,A -85,B 0,C 180,E1 -16526.122,E2 -16526.122} C_VEL
LIN {X 0,Y 298.301,Z 801.377,A -85,B 0,C 180,E1 -16526.345,E2 -16526.345} C_VEL
LIN {X 0,Y 297.714,Z 815.701,A -85,B 0,C 180,E1 -16527.225,E2 -16527.225} C_VEL
LIN {X 0,Y 297.086,Z 826.37,A -85,B 0,C 180,E1 -16528.101,E2 -16528.101} C_VEL
LIN {X 0,Y 296.372,Z 836.63,A -85,B 0,C 180,E1 -16529.149,E2 -16529.149} C_VEL
LIN {X 0,Y 295.693,Z 845.579,A -85,B 0,C 180,E1 -16530.254,E2 -16530.254} C_VEL
LIN {X 0,Y 294.979,Z 854.334,A -85,B 0,C 180,E1 -16531.542,E2 -16531.542} C_VEL
LIN {X 0,Y 294.265,Z 862.734,A -85,B 0,C 180,E1 -16533.013,E2 -16533.013} C_VEL
LIN {X 0,Y 293.571,Z 869.833,A -85,B 0,C 180,E1 -16534.474,E2 -16534.474} C_VEL
LIN {X 0,Y 292.959,Z 875.914,A -85,B 0,C 180,E1 -16535.931,E2 -16535.931} C_VEL
LIN {X 0,Y 292.491,Z 882.256,A -85,B 0,C 180,E1 -16537.762,E2 -16537.762} C_VEL
LIN {X 0,Y 292.013,Z 888.065,A -85,B 0,C 180,E1 -16539.827,E2 -16539.827} C_VEL
LIN {X 0,Y 291.724,Z 892.389,A -85,B 0,C 180,E1 -16541.748,E2 -16541.748} C_VEL
LIN {X 0,Y 291.633,Z 895.076,A -85,B 0,C 180,E1 -16543.19,E2 -16543.19} C_VEL
LIN {X 0,Y 291.603,Z 897.102,A -85,B 0,C 180,E1 -16544.626,E2 -16544.626} C_VEL
LIN {X 0,Y 291.784,Z 899.877,A -85,B 0,C 180,E1 -16547.48,E2 -16547.48} C_VEL
LIN {X 0,Y 292.049,Z 900.548,A -85,B 0,C 180,E1 -16548.9,E2 -16548.9} C_VEL
LIN {X 0,Y 292.365,Z 900.807,A -85,B 0,C 180,E1 -16550.313,E2 -16550.313} C_VEL
LIN {X 0,Y 292.732,Z 900.56,A -85,B 0,C 180,E1 -16551.717,E2 -16551.717} C_VEL
LIN {X 0,Y 293.236,Z 899.903,A -85,B 0,C 180,E1 -16553.117,E2 -16553.117} C_VEL
LIN {X 0,Y 294.533,Z 897.231,A -85,B 0,C 180,E1 -16555.895,E2 -16555.895} C_VEL
LIN {X 0,Y 295.798,Z 893.647,A -85,B 0,C 180,E1 -16558.156,E2 -16558.156} C_VEL
LIN {X 0,Y 297.066,Z 889.711,A -85,B 0,C 180,E1 -16560,E2 -16560} C_VEL
LIN {X 0,Y 298.42,Z 885.171,A -85,B 0,C 180,E1 -16561.687,E2 -16561.687} C_VEL
LIN {X 0,Y 299.981,Z 879.607,A -85,B 0,C 180,E1 -16563.358,E2 -16563.358} C_VEL
LIN {X 0,Y 301.585,Z 872.912,A -85,B 0,C 180,E1 -16565.013,E2 -16565.013} C_VEL
LIN {X 0,Y 303.069,Z 866.613,A -85,B 0,C 180,E1 -16566.324,E2 -16566.324} C_VEL
LIN {X 0,Y 304.934,Z 857.118,A -85,B 0,C 180,E1 -16567.948,E2 -16567.948} C_VEL
LIN {X 0,Y 306.327,Z 849.198,A -85,B 0,C 180,E1 -16569.07,E2 -16569.07} C_VEL
LIN {X 0,Y 307.706,Z 839.631,A -85,B 0,C 180,E1 -16570.195,E2 -16570.195} C_VEL
LIN {X 0,Y 308.87,Z 829.627,A -85,B 0,C 180,E1 -16571.152,E2 -16571.152} C_VEL
LIN {X 0,Y 309.729,Z 820.473,A -85,B 0,C 180,E1 -16571.867,E2 -16571.867} C_VEL
LIN {X 0,Y 310.463,Z 810.227,A -85,B 0,C 180,E1 -16572.491,E2 -16572.491} C_VEL
LIN {X 0,Y 311.053,Z 795.964,A -85,B 0,C 180,E1 -16573.132,E2 -16573.132} C_VEL
LIN {X 0,Y 312.644,Z 769.281,A -85,B 0,C 180,E1 -16574.086,E2 -16574.086} C_VEL
LIN {X 0,Y 313.776,Z 752.608,A -85,B 0,C 180,E1 -16574.674,E2 -16574.674} C_VEL
LIN {X 0,Y 308.021,Z 741.505,A -85,B 0,C 180,E1 -16576.3,E2 -16576.3} C_VEL
LIN {X 0,Y 302.865,Z 733.297,A -85,B 0,C 180,E1 -16577.856,E2 -16577.856} C_VEL
LIN {X 0,Y 300.635,Z 729.954,A -85,B 0,C 180,E1 -16578.57,E2 -16578.57} C_VEL
LIN {X 0,Y 298.122,Z 726.138,A -85,B 0,C 180,E1 -16579.439,E2 -16579.439} C_VEL
LIN {X 0,Y 295.691,Z 722.977,A -85,B 0,C 180,E1 -16580.296,E2 -16580.296} C_VEL
LIN {X 0,Y 294.926,Z 721.478,A -85,B 0,C 180,E1 -16580.62,E2 -16580.62} C_VEL
LIN {X 0,Y 292.633,Z 719.43,A -85,B 0,C 180,E1 -16581.449,E2 -16581.449} C_VEL
LIN {X 0,Y 291.476,Z 716.717,A -85,B 0,C 180,E1 -16582.132,E2 -16582.132} C_VEL
LIN {X 0,Y 291.38,Z 716.218,A -85,B 0,C 180,E1 -16582.7,E2 -16582.7} C_VEL
LIN {X 0,Y 291.366,Z 716.19,A -85,B 0,C 180,E1 -16586.811,E2 -16586.811} C_VEL
LIN {X 0,Y 291.329,Z 716.194,A -85,B 0,C 180,E1 -16590.438,E2 -16590.438} C_VEL
LIN {X 0,Y 291.351,Z 716.194,A -85,B 0,C 180,E1 -16593.697,E2 -16593.697} C_VEL
LIN {X 0,Y 291.391,Z 716.186,A -85,B 0,C 180,E1 -16597.255,E2 -16597.255} C_VEL
LIN {X 0,Y 291.341,Z 716.192,A -85,B 0,C 180,E1 -16600.641,E2 -16600.641} C_VEL
LIN {X 0,Y 291.297,Z 716.2,A -85,B 0,C 180,E1 -16604.401,E2 -16604.401} C_VEL
LIN {X 0,Y 291.332,Z 716.195,A -85,B 0,C 180,E1 -16608.403,E2 -16608.403} C_VEL
LIN {X 0,Y 291.427,Z 716.441,A -85,B 0,C 180,E1 -16609.938,E2 -16609.938} C_VEL
LIN {X 0,Y 293.487,Z 724.475,A -85,B 0,C 180,E1 -16612.208,E2 -16612.208} C_VEL
LIN {X 0,Y 295.449,Z 731.987,A -85,B 0,C 180,E1 -16613.977,E2 -16613.977} C_VEL
LIN {X 0,Y 299.807,Z 745.808,A -85,B 0,C 180,E1 -16616.66,E2 -16616.66} C_VEL
LIN {X 0,Y 302.806,Z 754.485,A -85,B 0,C 180,E1 -16617.824,E2 -16617.824} C_VEL
LIN {X 0,Y 305.746,Z 777.326,A -85,B 0,C 180,E1 -16619.62,E2 -16619.62} C_VEL
LIN {X 0,Y 308.008,Z 802.021,A -85,B 0,C 180,E1 -16621.227,E2 -16621.227} C_VEL
LIN {X 0,Y 308.7,Z 814.541,A -85,B 0,C 180,E1 -16621.921,E2 -16621.921} C_VEL
LIN {X 0,Y 309.214,Z 836.058,A -85,B 0,C 180,E1 -16622.961,E2 -16622.961} C_VEL
LIN {X 0,Y 306.697,Z 874.033,A -85,B 0,C 180,E1 -16624.279,E2 -16624.279} C_VEL
LIN {X 0,Y 305.15,Z 887.93,A -85,B 0,C 180,E1 -16624.961,E2 -16624.961} C_VEL
LIN {X 0,Y 303.215,Z 901.053,A -85,B 0,C 180,E1 -16625.886,E2 -16625.886} C_VEL
LIN {X 0,Y 301.111,Z 912.982,A -85,B 0,C 180,E1 -16626.984,E2 -16626.984} C_VEL
LIN {X 0,Y 299.194,Z 922.866,A -85,B 0,C 180,E1 -16628.103,E2 -16628.103} C_VEL
LIN {X 0,Y 297.481,Z 931.283,A -85,B 0,C 180,E1 -16629.243,E2 -16629.243} C_VEL
LIN {X 0,Y 295.783,Z 939.537,A -85,B 0,C 180,E1 -16630.568,E2 -16630.568} C_VEL
LIN {X 0,Y 293.999,Z 948.24,A -85,B 0,C 180,E1 -16632.253,E2 -16632.253} C_VEL
LIN {X 0,Y 292.725,Z 955.052,A -85,B 0,C 180,E1 -16633.813,E2 -16633.813} C_VEL
LIN {X 0,Y 291.644,Z 961.917,A -85,B 0,C 180,E1 -16635.698,E2 -16635.698} C_VEL
LIN {X 0,Y 290.929,Z 967.242,A -85,B 0,C 180,E1 -16637.441,E2 -16637.441} C_VEL
LIN {X 0,Y 290.357,Z 975.808,A -85,B 0,C 180,E1 -16640.946,E2 -16640.946} C_VEL
LIN {X 0,Y 290.412,Z 979.866,A -85,B 0,C 180,E1 -16643.048,E2 -16643.048} C_VEL
LIN {X 0,Y 290.534,Z 981.947,A -85,B 0,C 180,E1 -16644.445,E2 -16644.445} C_VEL
LIN {X 0,Y 290.788,Z 983.603,A -85,B 0,C 180,E1 -16645.84,E2 -16645.84} C_VEL
LIN {X 0,Y 290.864,Z 984.797,A -85,B 0,C 180,E1 -16647.228,E2 -16647.228} C_VEL
LIN {X 0,Y 290.989,Z 985.527,A -85,B 0,C 180,E1 -16648.614,E2 -16648.614} C_VEL
LIN {X 0,Y 291.109,Z 985.835,A -85,B 0,C 180,E1 -16649.998,E2 -16649.998} C_VEL
LIN {X 0,Y 290.967,Z 985.694,A -85,B 0,C 180,E1 -16651.382,E2 -16651.382} C_VEL
LIN {X 0,Y 290.829,Z 985.142,A -85,B 0,C 180,E1 -16652.768,E2 -16652.768} C_VEL
LIN {X 0,Y 290.721,Z 984.134,A -85,B 0,C 180,E1 -16654.157,E2 -16654.157} C_VEL
LIN {X 0,Y 290.37,Z 980.828,A -85,B 0,C 180,E1 -16656.949,E2 -16656.949} C_VEL
LIN {X 0,Y 290.267,Z 977.163,A -85,B 0,C 180,E1 -16659.053,E2 -16659.053} C_VEL
LIN {X 0,Y 290.515,Z 972.426,A -85,B 0,C 180,E1 -16661.157,E2 -16661.157} C_VEL
LIN {X 0,Y 291.126,Z 966.497,A -85,B 0,C 180,E1 -16663.256,E2 -16663.256} C_VEL
LIN {X 0,Y 292.157,Z 959.185,A -85,B 0,C 180,E1 -16665.342,E2 -16665.342} C_VEL
LIN {X 0,Y 293.663,Z 950.129,A -85,B 0,C 180,E1 -16667.404,E2 -16667.404} C_VEL
LIN {X 0,Y 295.318,Z 940.939,A -85,B 0,C 180,E1 -16669.098,E2 -16669.098} C_VEL
LIN {X 0,Y 297.132,Z 930.911,A -85,B 0,C 180,E1 -16670.597,E2 -16670.597} C_VEL
LIN {X 0,Y 298.942,Z 919.92,A -85,B 0,C 180,E1 -16671.912,E2 -16671.912} C_VEL
LIN {X 0,Y 300.793,Z 907.7,A -85,B 0,C 180,E1 -16673.037,E2 -16673.037} C_VEL
LIN {X 0,Y 302.383,Z 895.018,A -85,B 0,C 180,E1 -16673.906,E2 -16673.906} C_VEL
LIN {X 0,Y 303.492,Z 881.626,A -85,B 0,C 180,E1 -16674.541,E2 -16674.541} C_VEL
LIN {X 0,Y 304.234,Z 862.924,A -85,B 0,C 180,E1 -16675.058,E2 -16675.058} C_VEL
LIN {X 0,Y 304.991,Z 832.642,A -85,B 0,C 180,E1 -16675.802,E2 -16675.802} C_VEL
LIN {X 0,Y 302.303,Z 802.167,A -85,B 0,C 180,E1 -16676.907,E2 -16676.907} C_VEL
LIN {X 0,Y 299.202,Z 777.242,A -85,B 0,C 180,E1 -16677.935,E2 -16677.935} C_VEL
LIN {X 0,Y 297.5,Z 766.179,A -85,B 0,C 180,E1 -16678.482,E2 -16678.482} C_VEL
LIN {X 0,Y 299.77,Z 751.433,A -85,B 0,C 180,E1 -16681.748,E2 -16681.748} C_VEL
LIN {X 0,Y 297.441,Z 739.367,A -85,B 0,C 180,E1 -16684.956,E2 -16684.956} C_VEL
LIN {X 0,Y 294.613,Z 727.72,A -85,B 0,C 180,E1 -16688.33,E2 -16688.33} C_VEL
LIN {X 0,Y 291.341,Z 716.329,A -85,B 0,C 180,E1 -16692.015,E2 -16692.015} C_VEL
LIN {X 0,Y 291.33,Z 716.185,A -85,B 0,C 180,E1 -16696.359,E2 -16696.359} C_VEL
LIN {X 0,Y 291.378,Z 716.175,A -85,B 0,C 180,E1 -16700.515,E2 -16700.515} C_VEL
LIN {X 0,Y 291.416,Z 716.181,A -85,B 0,C 180,E1 -16702.921,E2 -16702.921} C_VEL
LIN {X 0,Y 291.335,Z 716.19,A -85,B 0,C 180,E1 -16706.3,E2 -16706.3} C_VEL
LIN {X 0,Y 291.377,Z 716.19,A -85,B 0,C 180,E1 -16710.259,E2 -16710.259} C_VEL
LIN {X 0,Y 291.41,Z 716.183,A -85,B 0,C 180,E1 -16714.271,E2 -16714.271} C_VEL
LIN {X 0,Y 291.37,Z 716.192,A -85,B 0,C 180,E1 -16717.299,E2 -16717.299} C_VEL
LIN {X 0,Y 291.447,Z 716.181,A -85,B 0,C 180,E1 -16720.27,E2 -16720.27} C_VEL
LIN {X 0,Y 291.544,Z 716.168,A -85,B 0,C 180,E1 -16724.623,E2 -16724.623} C_VEL
LIN {X 0,Y 291.524,Z 716.171,A -85,B 0,C 180,E1 -16728.88,E2 -16728.88} C_VEL
LIN {X 0,Y 291.675,Z 716.141,A -85,B 0,C 180,E1 -16731.688,E2 -16731.688} C_VEL
LIN {X 0,Y 291.616,Z 716.155,A -85,B 0,C 180,E1 -16734.468,E2 -16734.468} C_VEL
LIN {X 0,Y 291.878,Z 716.125,A -85,B 0,C 180,E1 -16738.62,E2 -16738.62} C_VEL
LIN {X 0,Y 291.878,Z 716.123,A -85,B 0,C 180,E1 -16741.38,E2 -16741.38} C_VEL
LIN {X 0,Y 291.734,Z 716.145,A -85,B 0,C 180,E1 -16746.918,E2 -16746.918} C_VEL
LIN {X 0,Y 291.618,Z 716.157,A -85,B 0,C 180,E1 -16749.713,E2 -16749.713} C_VEL
LIN {X 0,Y 291.511,Z 716.172,A -85,B 0,C 180,E1 -16753.951,E2 -16753.951} C_VEL
LIN {X 0,Y 291.475,Z 716.173,A -85,B 0,C 180,E1 -16756.819,E2 -16756.819} C_VEL
LIN {X 0,Y 291.44,Z 716.179,A -85,B 0,C 180,E1 -16759.876,E2 -16759.876} C_VEL
LIN {X 0,Y 291.372,Z 716.17,A -85,B 0,C 180,E1 -16764.208,E2 -16764.208} C_VEL
LIN {X 0,Y 291.414,Z 716.178,A -85,B 0,C 180,E1 -16767.273,E2 -16767.273} C_VEL
LIN {X 0,Y 291.325,Z 716.2,A -85,B 0,C 180,E1 -16770.439,E2 -16770.439} C_VEL
LIN {X 0,Y 291.336,Z 716.188,A -85,B 0,C 180,E1 -16773.7,E2 -16773.7} C_VEL
LIN {X 0,Y 291.421,Z 716.357,A -85,B 0,C 180,E1 -16776.218,E2 -16776.218} C_VEL
LIN {X 0,Y 291.594,Z 717.199,A -85,B 0,C 180,E1 -16776.461,E2 -16776.461} C_VEL
LIN {X 0,Y 293.149,Z 720.038,A -85,B 0,C 180,E1 -16776.771,E2 -16776.771} C_VEL
LIN {X 0,Y 301.747,Z 736.353,A -85,B 0,C 180,E1 -16778.273,E2 -16778.273} C_VEL
LIN {X 0,Y 307.236,Z 748.051,A -85,B 0,C 180,E1 -16779.199,E2 -16779.199} C_VEL
LIN {X 0,Y 306.153,Z 792.702,A -85,B 0,C 180,E1 -16780.317,E2 -16780.317} C_VEL
LIN {X 0,Y 306.025,Z 806.396,A -85,B 0,C 180,E1 -16780.779,E2 -16780.779} C_VEL
LIN {X 0,Y 305.606,Z 818.682,A -85,B 0,C 180,E1 -16781.447,E2 -16781.447} C_VEL
LIN {X 0,Y 304.839,Z 829.807,A -85,B 0,C 180,E1 -16782.274,E2 -16782.274} C_VEL
LIN {X 0,Y 303.618,Z 841.734,A -85,B 0,C 180,E1 -16783.43,E2 -16783.43} C_VEL
LIN {X 0,Y 302.235,Z 852.905,A -85,B 0,C 180,E1 -16784.831,E2 -16784.831} C_VEL
LIN {X 0,Y 300.649,Z 863.077,A -85,B 0,C 180,E1 -16786.441,E2 -16786.441} C_VEL
LIN {X 0,Y 299.201,Z 871.011,A -85,B 0,C 180,E1 -16787.979,E2 -16787.979} C_VEL
LIN {X 0,Y 297.617,Z 879.252,A -85,B 0,C 180,E1 -16789.951,E2 -16789.951} C_VEL
LIN {X 0,Y 296.274,Z 885.822,A -85,B 0,C 180,E1 -16791.924,E2 -16791.924} C_VEL
LIN {X 0,Y 294.882,Z 891.6,A -85,B 0,C 180,E1 -16794.129,E2 -16794.129} C_VEL
LIN {X 0,Y 293.683,Z 896.457,A -85,B 0,C 180,E1 -16796.608,E2 -16796.608} C_VEL
LIN {X 0,Y 293.111,Z 898.719,A -85,B 0,C 180,E1 -16798.166,E2 -16798.166} C_VEL
LIN {X 0,Y 292.678,Z 900.5,A -85,B 0,C 180,E1 -16799.822,E2 -16799.822} C_VEL
LIN {X 0,Y 292.338,Z 901.595,A -85,B 0,C 180,E1 -16801.264,E2 -16801.264} C_VEL
LIN {X 0,Y 292.065,Z 902.276,A -85,B 0,C 180,E1 -16802.916,E2 -16802.916} C_VEL
LIN {X 0,Y 291.921,Z 902.447,A -85,B 0,C 180,E1 -16804.322,E2 -16804.322} C_VEL
LIN {X 0,Y 291.861,Z 902.007,A -85,B 0,C 180,E1 -16806.213,E2 -16806.213} C_VEL
LIN {X 0,Y 292.078,Z 900.207,A -85,B 0,C 180,E1 -16808.845,E2 -16808.845} C_VEL
LIN {X 0,Y 292.505,Z 897.503,A -85,B 0,C 180,E1 -16811.075,E2 -16811.075} C_VEL
LIN {X 0,Y 293.244,Z 893.284,A -85,B 0,C 180,E1 -16813.469,E2 -16813.469} C_VEL
LIN {X 0,Y 294.037,Z 888.641,A -85,B 0,C 180,E1 -16815.467,E2 -16815.467} C_VEL
LIN {X 0,Y 295.076,Z 882.283,A -85,B 0,C 180,E1 -16817.624,E2 -16817.624} C_VEL
LIN {X 0,Y 296.345,Z 874.365,A -85,B 0,C 180,E1 -16819.757,E2 -16819.757} C_VEL
LIN {X 0,Y 297.53,Z 866.237,A -85,B 0,C 180,E1 -16821.512,E2 -16821.512} C_VEL
LIN {X 0,Y 298.896,Z 856.287,A -85,B 0,C 180,E1 -16823.25,E2 -16823.25} C_VEL
LIN {X 0,Y 300.219,Z 845.241,A -85,B 0,C 180,E1 -16824.797,E2 -16824.797} C_VEL
LIN {X 0,Y 301.308,Z 834.43,A -85,B 0,C 180,E1 -16825.989,E2 -16825.989} C_VEL
LIN {X 0,Y 302.243,Z 821.567,A -85,B 0,C 180,E1 -16827.086,E2 -16827.086} C_VEL
LIN {X 0,Y 302.77,Z 809.148,A -85,B 0,C 180,E1 -16827.866,E2 -16827.866} C_VEL
LIN {X 0,Y 303.002,Z 796.285,A -85,B 0,C 180,E1 -16828.397,E2 -16828.397} C_VEL
LIN {X 0,Y 303.889,Z 746.729,A -85,B 0,C 180,E1 -16829.634,E2 -16829.634} C_VEL
LIN {X 0,Y 303.816,Z 744.662,A -85,B 0,C 180,E1 -16829.694,E2 -16829.694} C_VEL
LIN {X 0,Y 297.588,Z 729.321,A -85,B 0,C 180,E1 -16830.624,E2 -16830.624} C_VEL
LIN {X 0,Y 292.071,Z 717.196,A -85,B 0,C 180,E1 -16831.467,E2 -16831.467} C_VEL
LIN {X 0,Y 291.845,Z 716.265,A -85,B 0,C 180,E1 -16831.727,E2 -16831.727} C_VEL
LIN {X 0,Y 291.69,Z 716.145,A -85,B 0,C 180,E1 -16836.921,E2 -16836.921} C_VEL
LIN {X 0,Y 291.572,Z 716.162,A -85,B 0,C 180,E1 -16839.716,E2 -16839.716} C_VEL
LIN {X 0,Y 291.519,Z 716.165,A -85,B 0,C 180,E1 -16843.952,E2 -16843.952} C_VEL
LIN {X 0,Y 291.431,Z 716.183,A -85,B 0,C 180,E1 -16846.823,E2 -16846.823} C_VEL
LIN {X 0,Y 291.397,Z 716.169,A -85,B 0,C 180,E1 -16849.844,E2 -16849.844} C_VEL
LIN {X 0,Y 291.34,Z 716.193,A -85,B 0,C 180,E1 -16854.213,E2 -16854.213} C_VEL
LIN {X 0,Y 291.334,Z 716.173,A -85,B 0,C 180,E1 -16857.283,E2 -16857.283} C_VEL
LIN {X 0,Y 291.307,Z 716.198,A -85,B 0,C 180,E1 -16860.442,E2 -16860.442} C_VEL
LIN {X 0,Y 291.35,Z 716.167,A -85,B 0,C 180,E1 -16863.7,E2 -16863.7} C_VEL
LIN {X 0,Y 291.359,Z 716.177,A -85,B 0,C 180,E1 -16867.249,E2 -16867.249} C_VEL
LIN {X 0,Y 291.301,Z 716.197,A -85,B 0,C 180,E1 -16870.65,E2 -16870.65} C_VEL
LIN {X 0,Y 291.288,Z 716.2,A -85,B 0,C 180,E1 -16874.405,E2 -16874.405} C_VEL
LIN {X 0,Y 291.301,Z 716.198,A -85,B 0,C 180,E1 -16878.413,E2 -16878.413} C_VEL
LIN {X 0,Y 291.342,Z 716.195,A -85,B 0,C 180,E1 -16881.156,E2 -16881.156} C_VEL
LIN {X 0,Y 291.414,Z 716.336,A -85,B 0,C 180,E1 -16882.861,E2 -16882.861} C_VEL
LIN {X 0,Y 291.617,Z 717.211,A -85,B 0,C 180,E1 -16883.086,E2 -16883.086} C_VEL
LIN {X 0,Y 299.861,Z 740.565,A -85,B 0,C 180,E1 -16884.342,E2 -16884.342} C_VEL
LIN {X 0,Y 298.422,Z 793.902,A -85,B 0,C 180,E1 -16886.016,E2 -16886.016} C_VEL
LIN {X 0,Y 298.301,Z 801.377,A -85,B 0,C 180,E1 -16886.345,E2 -16886.345} C_VEL
LIN {X 0,Y 297.331,Z 807.069,A -85,B 0,C 180,E1 -16886.598,E2 -16886.598} C_VEL
LIN {X 0,Y 294.098,Z 816.135,A -85,B 0,C 180,E1 -16887.069,E2 -16887.069} C_VEL
LIN {X 0,Y 290.82,Z 824.975,A -85,B 0,C 180,E1 -16887.67,E2 -16887.67} C_VEL
LIN {X 0,Y 289.92,Z 830.27,A -85,B 0,C 180,E1 -16888.161,E2 -16888.161} C_VEL
LIN {X 0,Y 289.306,Z 839.094,A -85,B 0,C 180,E1 -16889.125,E2 -16889.125} C_VEL
LIN {X 0,Y 288.555,Z 847.776,A -85,B 0,C 180,E1 -16890.247,E2 -16890.247} C_VEL
LIN {X 0,Y 287.882,Z 856.013,A -85,B 0,C 180,E1 -16891.509,E2 -16891.509} C_VEL
LIN {X 0,Y 287.316,Z 862.751,A -85,B 0,C 180,E1 -16892.7,E2 -16892.7} C_VEL
LIN {X 0,Y 286.612,Z 870.034,A -85,B 0,C 180,E1 -16894.199,E2 -16894.199} C_VEL
LIN {X 0,Y 285.859,Z 877.595,A -85,B 0,C 180,E1 -16896.067,E2 -16896.067} C_VEL
LIN {X 0,Y 285.352,Z 883.846,A -85,B 0,C 180,E1 -16897.938,E2 -16897.938} C_VEL
LIN {X 0,Y 284.957,Z 888.962,A -85,B 0,C 180,E1 -16899.8,E2 -16899.8} C_VEL
LIN {X 0,Y 284.733,Z 892.425,A -85,B 0,C 180,E1 -16901.284,E2 -16901.284} C_VEL
LIN {X 0,Y 284.565,Z 896.417,A -85,B 0,C 180,E1 -16903.499,E2 -16903.499} C_VEL
LIN {X 0,Y 284.576,Z 899.275,A -85,B 0,C 180,E1 -16905.702,E2 -16905.702} C_VEL
LIN {X 0,Y 284.704,Z 900.628,A -85,B 0,C 180,E1 -16907.163,E2 -16907.163} C_VEL
LIN {X 0,Y 284.987,Z 901.507,A -85,B 0,C 180,E1 -16908.621,E2 -16908.621} C_VEL
LIN {X 0,Y 285.312,Z 901.921,A -85,B 0,C 180,E1 -16910.176,E2 -16910.176} C_VEL
LIN {X 0,Y 285.672,Z 901.893,A -85,B 0,C 180,E1 -16911.511,E2 -16911.511} C_VEL
LIN {X 0,Y 286.802,Z 900.445,A -85,B 0,C 180,E1 -16914.375,E2 -16914.375} C_VEL
LIN {X 0,Y 287.532,Z 899.146,A -85,B 0,C 180,E1 -16915.795,E2 -16915.795} C_VEL
LIN {X 0,Y 288.448,Z 896.946,A -85,B 0,C 180,E1 -16917.423,E2 -16917.423} C_VEL
LIN {X 0,Y 290.169,Z 892.267,A -85,B 0,C 180,E1 -16920,E2 -16920} C_VEL
LIN {X 0,Y 292.193,Z 885.922,A -85,B 0,C 180,E1 -16922.412,E2 -16922.412} C_VEL
LIN {X 0,Y 293.855,Z 880.325,A -85,B 0,C 180,E1 -16924.114,E2 -16924.114} C_VEL
LIN {X 0,Y 295.241,Z 875.109,A -85,B 0,C 180,E1 -16925.464,E2 -16925.464} C_VEL
LIN {X 0,Y 297.172,Z 867.186,A -85,B 0,C 180,E1 -16927.132,E2 -16927.132} C_VEL
LIN {X 0,Y 298.774,Z 859.803,A -85,B 0,C 180,E1 -16928.431,E2 -16928.431} C_VEL
LIN {X 0,Y 300.333,Z 851.455,A -85,B 0,C 180,E1 -16929.668,E2 -16929.668} C_VEL
LIN {X 0,Y 301.933,Z 841.365,A -85,B 0,C 180,E1 -16930.901,E2 -16930.901} C_VEL
LIN {X 0,Y 303.215,Z 831.569,A -85,B 0,C 180,E1 -16931.871,E2 -16931.871} C_VEL
LIN {X 0,Y 304.154,Z 822.122,A -85,B 0,C 180,E1 -16932.633,E2 -16932.633} C_VEL
LIN {X 0,Y 304.966,Z 811.692,A -85,B 0,C 180,E1 -16933.281,E2 -16933.281} C_VEL
LIN {X 0,Y 305.57,Z 798.416,A -85,B 0,C 180,E1 -16933.899,E2 -16933.899} C_VEL
LIN {X 0,Y 307.291,Z 771.521,A -85,B 0,C 180,E1 -16934.908,E2 -16934.908} C_VEL
LIN {X 0,Y 308.511,Z 755.484,A -85,B 0,C 180,E1 -16935.487,E2 -16935.487} C_VEL
LIN {X 0,Y 303.535,Z 745.823,A -85,B 0,C 180,E1 -16936.989,E2 -16936.989} C_VEL
LIN {X 0,Y 298.877,Z 738.191,A -85,B 0,C 180,E1 -16938.488,E2 -16938.488} C_VEL
LIN {X 0,Y 296.179,Z 734.134,A -85,B 0,C 180,E1 -16939.432,E2 -16939.432} C_VEL
LIN {X 0,Y 294.529,Z 731.625,A -85,B 0,C 180,E1 -16940.026,E2 -16940.026} C_VEL
LIN {X 0,Y 292.188,Z 728.148,A -85,B 0,C 180,E1 -16940.948,E2 -16940.948} C_VEL
LIN {X 0,Y 289.131,Z 724.504,A -85,B 0,C 180,E1 -16942.183,E2 -16942.183} C_VEL
LIN {X 0,Y 288.195,Z 722.57,A -85,B 0,C 180,E1 -16942.663,E2 -16942.663} C_VEL
LIN {X 0,Y 285.759,Z 720.499,A -85,B 0,C 180,E1 -16943.715,E2 -16943.715} C_VEL
LIN {X 0,Y 284.454,Z 717.806,A -85,B 0,C 180,E1 -16944.549,E2 -16944.549} C_VEL
LIN {X 0,Y 284.33,Z 717.105,A -85,B 0,C 180,E1 -16945.238,E2 -16945.238} C_VEL
LIN {X 0,Y 284.299,Z 717.072,A -85,B 0,C 180,E1 -16948.014,E2 -16948.014} C_VEL
LIN {X 0,Y 284.294,Z 717.072,A -85,B 0,C 180,E1 -16951.274,E2 -16951.274} C_VEL
LIN {X 0,Y 284.349,Z 717.065,A -85,B 0,C 180,E1 -16955.347,E2 -16955.347} C_VEL
LIN {X 0,Y 284.327,Z 717.068,A -85,B 0,C 180,E1 -16958.167,E2 -16958.167} C_VEL
LIN {X 0,Y 284.276,Z 717.076,A -85,B 0,C 180,E1 -16962.123,E2 -16962.123} C_VEL
LIN {X 0,Y 284.288,Z 717.135,A -85,B 0,C 180,E1 -16966.641,E2 -16966.641} C_VEL
LIN {X 0,Y 284.382,Z 717.612,A -85,B 0,C 180,E1 -16967.451,E2 -16967.451} C_VEL
LIN {X 0,Y 285.006,Z 719.426,A -85,B 0,C 180,E1 -16968.254,E2 -16968.254} C_VEL
LIN {X 0,Y 286.733,Z 721.564,A -85,B 0,C 180,E1 -16969.449,E2 -16969.449} C_VEL
LIN {X 0,Y 287.609,Z 723.955,A -85,B 0,C 180,E1 -16970.248,E2 -16970.248} C_VEL
LIN {X 0,Y 290.223,Z 733.681,A -85,B 0,C 180,E1 -16972.74,E2 -16972.74} C_VEL
LIN {X 0,Y 293.092,Z 743.826,A -85,B 0,C 180,E1 -16974.843,E2 -16974.843} C_VEL
LIN {X 0,Y 296.386,Z 752.167,A -85,B 0,C 180,E1 -16976.229,E2 -16976.229} C_VEL
LIN {X 0,Y 298.246,Z 758.151,A -85,B 0,C 180,E1 -16977.023,E2 -16977.023} C_VEL
LIN {X 0,Y 300.599,Z 778.23,A -85,B 0,C 180,E1 -16978.659,E2 -16978.659} C_VEL
LIN {X 0,Y 302.51,Z 800.42,A -85,B 0,C 180,E1 -16980.195,E2 -16980.195} C_VEL
LIN {X 0,Y 303.275,Z 814.682,A -85,B 0,C 180,E1 -16981.033,E2 -16981.033} C_VEL
LIN {X 0,Y 303.66,Z 836.839,A -85,B 0,C 180,E1 -16982.149,E2 -16982.149} C_VEL
LIN {X 0,Y 301.178,Z 872.041,A -85,B 0,C 180,E1 -16983.409,E2 -16983.409} C_VEL
LIN {X 0,Y 299.698,Z 884.339,A -85,B 0,C 180,E1 -16984.007,E2 -16984.007} C_VEL
LIN {X 0,Y 297.48,Z 899.055,A -85,B 0,C 180,E1 -16985.018,E2 -16985.018} C_VEL
LIN {X 0,Y 295.232,Z 911.107,A -85,B 0,C 180,E1 -16986.127,E2 -16986.127} C_VEL
LIN {X 0,Y 293.15,Z 921.026,A -85,B 0,C 180,E1 -16987.256,E2 -16987.256} C_VEL
LIN {X 0,Y 291.106,Z 930.535,A -85,B 0,C 180,E1 -16988.581,E2 -16988.581} C_VEL
LIN {X 0,Y 289.467,Z 937.754,A -85,B 0,C 180,E1 -16989.757,E2 -16989.757} C_VEL
LIN {X 0,Y 287.558,Z 946.545,A -85,B 0,C 180,E1 -16991.473,E2 -16991.473} C_VEL
LIN {X 0,Y 286.069,Z 954.002,A -85,B 0,C 180,E1 -16993.225,E2 -16993.225} C_VEL
LIN {X 0,Y 284.937,Z 960.304,A -85,B 0,C 180,E1 -16994.988,E2 -16994.988} C_VEL
LIN {X 0,Y 283.95,Z 966.595,A -85,B 0,C 180,E1 -16997.127,E2 -16997.127} C_VEL
LIN {X 0,Y 283.397,Z 971.697,A -85,B 0,C 180,E1 -16999.279,E2 -16999.279} C_VEL
LIN {X 0,Y 283.35,Z 977.636,A -85,B 0,C 180,E1 -17002.229,E2 -17002.229} C_VEL
LIN {X 0,Y 283.456,Z 980.86,A -85,B 0,C 180,E1 -17004.306,E2 -17004.306} C_VEL
LIN {X 0,Y 283.718,Z 982.532,A -85,B 0,C 180,E1 -17005.736,E2 -17005.736} C_VEL
LIN {X 0,Y 283.819,Z 983.747,A -85,B 0,C 180,E1 -17007.159,E2 -17007.159} C_VEL
LIN {X 0,Y 283.951,Z 984.498,A -85,B 0,C 180,E1 -17008.58,E2 -17008.58} C_VEL
LIN {X 0,Y 284.079,Z 984.818,A -85,B 0,C 180,E1 -17009.998,E2 -17009.998} C_VEL
LIN {X 0,Y 283.926,Z 984.686,A -85,B 0,C 180,E1 -17011.416,E2 -17011.416} C_VEL
LIN {X 0,Y 283.777,Z 984.145,A -85,B 0,C 180,E1 -17012.837,E2 -17012.837} C_VEL
LIN {X 0,Y 283.64,Z 983.153,A -85,B 0,C 180,E1 -17014.261,E2 -17014.261} C_VEL
LIN {X 0,Y 283.291,Z 979.865,A -85,B 0,C 180,E1 -17017.123,E2 -17017.123} C_VEL
LIN {X 0,Y 283.202,Z 976.221,A -85,B 0,C 180,E1 -17019.28,E2 -17019.28} C_VEL
LIN {X 0,Y 283.472,Z 971.507,A -85,B 0,C 180,E1 -17021.438,E2 -17021.438} C_VEL
LIN {X 0,Y 284.149,Z 965.608,A -85,B 0,C 180,E1 -17023.587,E2 -17023.587} C_VEL
LIN {X 0,Y 285.085,Z 959.638,A -85,B 0,C 180,E1 -17025.365,E2 -17025.365} C_VEL
LIN {X 0,Y 285.678,Z 955.756,A -85,B 0,C 180,E1 -17026.373,E2 -17026.373} C_VEL
LIN {X 0,Y 287.121,Z 947.665,A -85,B 0,C 180,E1 -17028.183,E2 -17028.183} C_VEL
LIN {X 0,Y 288.953,Z 938.214,A -85,B 0,C 180,E1 -17029.906,E2 -17029.906} C_VEL
LIN {X 0,Y 290.947,Z 927.775,A -85,B 0,C 180,E1 -17031.427,E2 -17031.427} C_VEL
LIN {X 0,Y 292.928,Z 916.275,A -85,B 0,C 180,E1 -17032.758,E2 -17032.758} C_VEL
LIN {X 0,Y 294.733,Z 904.402,A -85,B 0,C 180,E1 -17033.819,E2 -17033.819} C_VEL
LIN {X 0,Y 296.284,Z 891.451,A -85,B 0,C 180,E1 -17034.664,E2 -17034.664} C_VEL
LIN {X 0,Y 297.352,Z 878.163,A -85,B 0,C 180,E1 -17035.254,E2 -17035.254} C_VEL
LIN {X 0,Y 298.69,Z 833.215,A -85,B 0,C 180,E1 -17036.417,E2 -17036.417} C_VEL
LIN {X 0,Y 296.108,Z 803.168,A -85,B 0,C 180,E1 -17037.535,E2 -17037.535} C_VEL
LIN {X 0,Y 293.192,Z 779.207,A -85,B 0,C 180,E1 -17038.562,E2 -17038.562} C_VEL
LIN {X 0,Y 291.034,Z 765.017,A -85,B 0,C 180,E1 -17039.285,E2 -17039.285} C_VEL
LIN {X 0,Y 292.926,Z 753.606,A -85,B 0,C 180,E1 -17041.856,E2 -17041.856} C_VEL
LIN {X 0,Y 291.829,Z 746.949,A -85,B 0,C 180,E1 -17043.632,E2 -17043.632} C_VEL
LIN {X 0,Y 289.448,Z 736.019,A -85,B 0,C 180,E1 -17046.749,E2 -17046.749} C_VEL
LIN {X 0,Y 286.781,Z 725.754,A -85,B 0,C 180,E1 -17049.933,E2 -17049.933} C_VEL
LIN {X 0,Y 284.288,Z 717.162,A -85,B 0,C 180,E1 -17052.909,E2 -17052.909} C_VEL
LIN {X 0,Y 284.277,Z 717.063,A -85,B 0,C 180,E1 -17056.193,E2 -17056.193} C_VEL
LIN {X 0,Y 284.303,Z 717.055,A -85,B 0,C 180,E1 -17060.021,E2 -17060.021} C_VEL
LIN {X 0,Y 284.341,Z 717.053,A -85,B 0,C 180,E1 -17063.615,E2 -17063.615} C_VEL
LIN {X 0,Y 284.298,Z 717.074,A -85,B 0,C 180,E1 -17067.188,E2 -17067.188} C_VEL
LIN {X 0,Y 284.349,Z 717.066,A -85,B 0,C 180,E1 -17070.375,E2 -17070.375} C_VEL
LIN {X 0,Y 284.37,Z 717.064,A -85,B 0,C 180,E1 -17073.586,E2 -17073.586} C_VEL
LIN {X 0,Y 284.355,Z 717.064,A -85,B 0,C 180,E1 -17076.706,E2 -17076.706} C_VEL
LIN {X 0,Y 284.393,Z 717.059,A -85,B 0,C 180,E1 -17081.261,E2 -17081.261} C_VEL
LIN {X 0,Y 284.481,Z 717.049,A -85,B 0,C 180,E1 -17084.458,E2 -17084.458} C_VEL
LIN {X 0,Y 284.476,Z 717.049,A -85,B 0,C 180,E1 -17088.601,E2 -17088.601} C_VEL
LIN {X 0,Y 284.627,Z 717.018,A -85,B 0,C 180,E1 -17091.48,E2 -17091.48} C_VEL
LIN {X 0,Y 284.586,Z 717.032,A -85,B 0,C 180,E1 -17094.331,E2 -17094.331} C_VEL
LIN {X 0,Y 284.844,Z 717.001,A -85,B 0,C 180,E1 -17098.586,E2 -17098.586} C_VEL
LIN {X 0,Y 284.844,Z 716.999,A -85,B 0,C 180,E1 -17101.414,E2 -17101.414} C_VEL
LIN {X 0,Y 284.686,Z 717.022,A -85,B 0,C 180,E1 -17107.091,E2 -17107.091} C_VEL
LIN {X 0,Y 284.555,Z 717.037,A -85,B 0,C 180,E1 -17109.956,E2 -17109.956} C_VEL
LIN {X 0,Y 284.471,Z 717.051,A -85,B 0,C 180,E1 -17114.304,E2 -17114.304} C_VEL
LIN {X 0,Y 284.412,Z 717.057,A -85,B 0,C 180,E1 -17117.249,E2 -17117.249} C_VEL
LIN {X 0,Y 284.366,Z 717.062,A -85,B 0,C 180,E1 -17120.243,E2 -17120.243} C_VEL
LIN {X 0,Y 284.33,Z 717.053,A -85,B 0,C 180,E1 -17124.848,E2 -17124.848} C_VEL
LIN {X 0,Y 284.321,Z 717.054,A -85,B 0,C 180,E1 -17128.012,E2 -17128.012} C_VEL
LIN {X 0,Y 284.285,Z 717.072,A -85,B 0,C 180,E1 -17131.276,E2 -17131.276} C_VEL
LIN {X 0,Y 284.371,Z 717.209,A -85,B 0,C 180,E1 -17135.292,E2 -17135.292} C_VEL
LIN {X 0,Y 284.601,Z 718.283,A -85,B 0,C 180,E1 -17135.587,E2 -17135.587} C_VEL
LIN {X 0,Y 292.184,Z 731.927,A -85,B 0,C 180,E1 -17137.01,E2 -17137.01} C_VEL
LIN {X 0,Y 300.327,Z 748.488,A -85,B 0,C 180,E1 -17138.46,E2 -17138.46} C_VEL
LIN {X 0,Y 301.063,Z 750.147,A -85,B 0,C 180,E1 -17138.589,E2 -17138.589} C_VEL
LIN {X 0,Y 299.926,Z 792.598,A -85,B 0,C 180,E1 -17139.668,E2 -17139.668} C_VEL
LIN {X 0,Y 299.769,Z 807.495,A -85,B 0,C 180,E1 -17140.173,E2 -17140.173} C_VEL
LIN {X 0,Y 299.367,Z 818.875,A -85,B 0,C 180,E1 -17140.795,E2 -17140.795} C_VEL
LIN {X 0,Y 298.465,Z 831.41,A -85,B 0,C 180,E1 -17141.745,E2 -17141.745} C_VEL
LIN {X 0,Y 297.253,Z 842.726,A -85,B 0,C 180,E1 -17142.87,E2 -17142.87} C_VEL
LIN {X 0,Y 295.93,Z 852.921,A -85,B 0,C 180,E1 -17144.158,E2 -17144.158} C_VEL
LIN {X 0,Y 294.313,Z 863.051,A -85,B 0,C 180,E1 -17145.757,E2 -17145.757} C_VEL
LIN {X 0,Y 292.802,Z 871.08,A -85,B 0,C 180,E1 -17147.31,E2 -17147.31} C_VEL
LIN {X 0,Y 291.098,Z 879.475,A -85,B 0,C 180,E1 -17149.321,E2 -17149.321} C_VEL
LIN {X 0,Y 289.626,Z 886.198,A -85,B 0,C 180,E1 -17151.332,E2 -17151.332} C_VEL
LIN {X 0,Y 288.18,Z 892.152,A -85,B 0,C 180,E1 -17153.591,E2 -17153.591} C_VEL
LIN {X 0,Y 287.029,Z 896.467,A -85,B 0,C 180,E1 -17155.728,E2 -17155.728} C_VEL
LIN {X 0,Y 286.407,Z 898.939,A -85,B 0,C 180,E1 -17157.33,E2 -17157.33} C_VEL
LIN {X 0,Y 285.767,Z 901.309,A -85,B 0,C 180,E1 -17159.404,E2 -17159.404} C_VEL
LIN {X 0,Y 285.202,Z 903.083,A -85,B 0,C 180,E1 -17162.085,E2 -17162.085} C_VEL
LIN {X 0,Y 284.95,Z 903.441,A -85,B 0,C 180,E1 -17163.646,E2 -17163.646} C_VEL
LIN {X 0,Y 284.845,Z 903.129,A -85,B 0,C 180,E1 -17165.911,E2 -17165.911} C_VEL
LIN {X 0,Y 284.965,Z 901.719,A -85,B 0,C 180,E1 -17168.291,E2 -17168.291} C_VEL
LIN {X 0,Y 285.217,Z 900.217,A -85,B 0,C 180,E1 -17169.822,E2 -17169.822} C_VEL
LIN {X 0,Y 285.773,Z 897.061,A -85,B 0,C 180,E1 -17172.099,E2 -17172.099} C_VEL
LIN {X 0,Y 286.522,Z 892.771,A -85,B 0,C 180,E1 -17174.349,E2 -17174.349} C_VEL
LIN {X 0,Y 287.678,Z 886.136,A -85,B 0,C 180,E1 -17176.942,E2 -17176.942} C_VEL
LIN {X 0,Y 288.913,Z 878.913,A -85,B 0,C 180,E1 -17179.136,E2 -17179.136} C_VEL
LIN {X 0,Y 290.083,Z 871.528,A -85,B 0,C 180,E1 -17180.942,E2 -17180.942} C_VEL
LIN {X 0,Y 291.526,Z 861.842,A -85,B 0,C 180,E1 -17182.852,E2 -17182.852} C_VEL
LIN {X 0,Y 292.867,Z 851.517,A -85,B 0,C 180,E1 -17184.494,E2 -17184.494} C_VEL
LIN {X 0,Y 294.149,Z 840.411,A -85,B 0,C 180,E1 -17185.892,E2 -17185.892} C_VEL
LIN {X 0,Y 295.249,Z 828.04,A -85,B 0,C 180,E1 -17187.103,E2 -17187.103} C_VEL
LIN {X 0,Y 295.94,Z 816.163,A -85,B 0,C 180,E1 -17187.986,E2 -17187.986} C_VEL
LIN {X 0,Y 296.364,Z 803.634,A -85,B 0,C 180,E1 -17188.643,E2 -17188.643} C_VEL
LIN {X 0,Y 296.519,Z 788.617,A -85,B 0,C 180,E1 -17189.12,E2 -17189.12} C_VEL
LIN {X 0,Y 297.289,Z 746.507,A -85,B 0,C 180,E1 -17190.184,E2 -17190.184} C_VEL
LIN {X 0,Y 291.757,Z 732.756,A -85,B 0,C 180,E1 -17191.041,E2 -17191.041} C_VEL
LIN {X 0,Y 284.943,Z 717.94,A -85,B 0,C 180,E1 -17192.12,E2 -17192.12} C_VEL
LIN {X 0,Y 284.748,Z 717.082,A -85,B 0,C 180,E1 -17192.433,E2 -17192.433} C_VEL
LIN {X 0,Y 284.645,Z 717.022,A -85,B 0,C 180,E1 -17197.093,E2 -17197.093} C_VEL
LIN {X 0,Y 284.518,Z 717.038,A -85,B 0,C 180,E1 -17199.959,E2 -17199.959} C_VEL
LIN {X 0,Y 284.468,Z 717.04,A -85,B 0,C 180,E1 -17204.306,E2 -17204.306} C_VEL
LIN {X 0,Y 284.334,Z 717.056,A -85,B 0,C 180,E1 -17208.745,E2 -17208.745} C_VEL
LIN {X 0,Y 284.315,Z 717.07,A -85,B 0,C 180,E1 -17213.3,E2 -17213.3} C_VEL
LIN {X 0,Y 284.292,Z 717.049,A -85,B 0,C 180,E1 -17217.131,E2 -17217.131} C_VEL
LIN {X 0,Y 284.279,Z 717.073,A -85,B 0,C 180,E1 -17220.085,E2 -17220.085} C_VEL
LIN {X 0,Y 284.311,Z 717.051,A -85,B 0,C 180,E1 -17222.947,E2 -17222.947} C_VEL
LIN {X 0,Y 284.325,Z 717.045,A -85,B 0,C 180,E1 -17226.389,E2 -17226.389} C_VEL
LIN {X 0,Y 284.288,Z 717.072,A -85,B 0,C 180,E1 -17230,E2 -17230} C_VEL
LIN {X 0,Y 284.24,Z 717.079,A -85,B 0,C 180,E1 -17234.188,E2 -17234.188} C_VEL
LIN {X 0,Y 284.246,Z 717.078,A -85,B 0,C 180,E1 -17238.119,E2 -17238.119} C_VEL
LIN {X 0,Y 284.332,Z 717.093,A -85,B 0,C 180,E1 -17242.278,E2 -17242.278} C_VEL
LIN {X 0,Y 284.433,Z 717.554,A -85,B 0,C 180,E1 -17242.615,E2 -17242.615} C_VEL
LIN {X 0,Y 285.068,Z 719.616,A -85,B 0,C 180,E1 -17242.812,E2 -17242.812} C_VEL
LIN {X 0,Y 292.886,Z 741.72,A -85,B 0,C 180,E1 -17244.012,E2 -17244.012} C_VEL
LIN {X 0,Y 291.522,Z 795.099,A -85,B 0,C 180,E1 -17245.752,E2 -17245.752} C_VEL
LIN {X 0,Y 291.176,Z 806.834,A -85,B 0,C 180,E1 -17246.331,E2 -17246.331} C_VEL
LIN {X 0,Y 290.712,Z 817.533,A -85,B 0,C 180,E1 -17247.047,E2 -17247.047} C_VEL
LIN {X 0,Y 290.089,Z 827.688,A -85,B 0,C 180,E1 -17247.908,E2 -17247.908} C_VEL
LIN {X 0,Y 289.92,Z 830.27,A -85,B 0,C 180,E1 -17248.161,E2 -17248.161} C_VEL
LIN {X 0,Y 288.938,Z 835.552,A -85,B 0,C 180,E1 -17248.668,E2 -17248.668} C_VEL
LIN {X 0,Y 285.559,Z 843.792,A -85,B 0,C 180,E1 -17249.52,E2 -17249.52} C_VEL
LIN {X 0,Y 282.07,Z 851.687,A -85,B 0,C 180,E1 -17250.514,E2 -17250.514} C_VEL
LIN {X 0,Y 280.938,Z 856.264,A -85,B 0,C 180,E1 -17251.237,E2 -17251.237} C_VEL
LIN {X 0,Y 280.189,Z 864.585,A -85,B 0,C 180,E1 -17252.756,E2 -17252.756} C_VEL
LIN {X 0,Y 279.484,Z 871.739,A -85,B 0,C 180,E1 -17254.292,E2 -17254.292} C_VEL
LIN {X 0,Y 278.84,Z 878.04,A -85,B 0,C 180,E1 -17255.874,E2 -17255.874} C_VEL
LIN {X 0,Y 278.329,Z 884.259,A -85,B 0,C 180,E1 -17257.743,E2 -17257.743} C_VEL
LIN {X 0,Y 278.037,Z 888.617,A -85,B 0,C 180,E1 -17259.275,E2 -17259.275} C_VEL
LIN {X 0,Y 277.665,Z 893.815,A -85,B 0,C 180,E1 -17261.555,E2 -17261.555} C_VEL
LIN {X 0,Y 277.534,Z 897.744,A -85,B 0,C 180,E1 -17263.826,E2 -17263.826} C_VEL
LIN {X 0,Y 277.53,Z 899.798,A -85,B 0,C 180,E1 -17265.331,E2 -17265.331} C_VEL
LIN {X 0,Y 277.888,Z 902.359,A -85,B 0,C 180,E1 -17268.327,E2 -17268.327} C_VEL
LIN {X 0,Y 278.294,Z 903.027,A -85,B 0,C 180,E1 -17270.041,E2 -17270.041} C_VEL
LIN {X 0,Y 278.598,Z 903.132,A -85,B 0,C 180,E1 -17271.294,E2 -17271.294} C_VEL
LIN {X 0,Y 279.762,Z 902.138,A -85,B 0,C 180,E1 -17274.233,E2 -17274.233} C_VEL
LIN {X 0,Y 281.33,Z 899.247,A -85,B 0,C 180,E1 -17277.136,E2 -17277.136} C_VEL
LIN {X 0,Y 282.235,Z 897.247,A -85,B 0,C 180,E1 -17278.573,E2 -17278.573} C_VEL
LIN {X 0,Y 283.795,Z 893.196,A -85,B 0,C 180,E1 -17280.709,E2 -17280.709} C_VEL
LIN {X 0,Y 285.693,Z 887.862,A -85,B 0,C 180,E1 -17282.82,E2 -17282.82} C_VEL
LIN {X 0,Y 287.463,Z 882.388,A -85,B 0,C 180,E1 -17284.557,E2 -17284.557} C_VEL
LIN {X 0,Y 289.316,Z 875.79,A -85,B 0,C 180,E1 -17286.276,E2 -17286.276} C_VEL
LIN {X 0,Y 291.285,Z 868.181,A -85,B 0,C 180,E1 -17287.905,E2 -17287.905} C_VEL
LIN {X 0,Y 293.089,Z 860.402,A -85,B 0,C 180,E1 -17289.291,E2 -17289.291} C_VEL
LIN {X 0,Y 294.691,Z 852.488,A -85,B 0,C 180,E1 -17290.477,E2 -17290.477} C_VEL
LIN {X 0,Y 296.245,Z 843.229,A -85,B 0,C 180,E1 -17291.633,E2 -17291.633} C_VEL
LIN {X 0,Y 297.617,Z 833.531,A -85,B 0,C 180,E1 -17292.617,E2 -17292.617} C_VEL
LIN {X 0,Y 298.691,Z 823.782,A -85,B 0,C 180,E1 -17293.435,E2 -17293.435} C_VEL
LIN {X 0,Y 299.601,Z 813.273,A -85,B 0,C 180,E1 -17294.114,E2 -17294.114} C_VEL
LIN {X 0,Y 300.318,Z 799.859,A -85,B 0,C 180,E1 -17294.762,E2 -17294.762} C_VEL
LIN {X 0,Y 302.173,Z 772.355,A -85,B 0,C 180,E1 -17295.822,E2 -17295.822} C_VEL
LIN {X 0,Y 303.261,Z 758.178,A -85,B 0,C 180,E1 -17296.365,E2 -17296.365} C_VEL
LIN {X 0,Y 298.41,Z 748.761,A -85,B 0,C 180,E1 -17297.952,E2 -17297.952} C_VEL
LIN {X 0,Y 293.484,Z 740.786,A -85,B 0,C 180,E1 -17299.696,E2 -17299.696} C_VEL
LIN {X 0,Y 290.954,Z 736.954,A -85,B 0,C 180,E1 -17300.68,E2 -17300.68} C_VEL
LIN {X 0,Y 288.374,Z 733.259,A -85,B 0,C 180,E1 -17301.736,E2 -17301.736} C_VEL
LIN {X 0,Y 286.057,Z 730.179,A -85,B 0,C 180,E1 -17302.774,E2 -17302.774} C_VEL
LIN {X 0,Y 285.147,Z 728.662,A -85,B 0,C 180,E1 -17303.225,E2 -17303.225} C_VEL
LIN {X 0,Y 282.8,Z 726.143,A -85,B 0,C 180,E1 -17304.378,E2 -17304.378} C_VEL
LIN {X 0,Y 281.425,Z 723.594,A -85,B 0,C 180,E1 -17305.205,E2 -17305.205} C_VEL
LIN {X 0,Y 278.676,Z 721.361,A -85,B 0,C 180,E1 -17306.795,E2 -17306.795} C_VEL
LIN {X 0,Y 277.354,Z 718.513,A -85,B 0,C 180,E1 -17308.054,E2 -17308.054} C_VEL
LIN {X 0,Y 277.271,Z 717.997,A -85,B 0,C 180,E1 -17308.789,E2 -17308.789} C_VEL
LIN {X 0,Y 277.248,Z 717.948,A -85,B 0,C 180,E1 -17312.163,E2 -17312.163} C_VEL
LIN {X 0,Y 277.315,Z 717.943,A -85,B 0,C 180,E1 -17315.806,E2 -17315.806} C_VEL
LIN {X 0,Y 277.244,Z 717.948,A -85,B 0,C 180,E1 -17319.326,E2 -17319.326} C_VEL
LIN {X 0,Y 277.262,Z 718.231,A -85,B 0,C 180,E1 -17323.307,E2 -17323.307} C_VEL
LIN {X 0,Y 278.135,Z 720.704,A -85,B 0,C 180,E1 -17325.033,E2 -17325.033} C_VEL
LIN {X 0,Y 280.01,Z 722.794,A -85,B 0,C 180,E1 -17326.709,E2 -17326.709} C_VEL
LIN {X 0,Y 281.879,Z 726.164,A -85,B 0,C 180,E1 -17328.416,E2 -17328.416} C_VEL
LIN {X 0,Y 283.022,Z 727.484,A -85,B 0,C 180,E1 -17329.183,E2 -17329.183} C_VEL
LIN {X 0,Y 284.608,Z 733.39,A -85,B 0,C 180,E1 -17330.896,E2 -17330.896} C_VEL
LIN {X 0,Y 286.741,Z 741.377,A -85,B 0,C 180,E1 -17332.784,E2 -17332.784} C_VEL
LIN {X 0,Y 292.232,Z 756.196,A -85,B 0,C 180,E1 -17335.43,E2 -17335.43} C_VEL
LIN {X 0,Y 293.744,Z 761.462,A -85,B 0,C 180,E1 -17336.153,E2 -17336.153} C_VEL
LIN {X 0,Y 295.829,Z 781.286,A -85,B 0,C 180,E1 -17337.827,E2 -17337.827} C_VEL
LIN {X 0,Y 297.511,Z 803.748,A -85,B 0,C 180,E1 -17339.416,E2 -17339.416} C_VEL
LIN {X 0,Y 298.01,Z 817.378,A -85,B 0,C 180,E1 -17340.239,E2 -17340.239} C_VEL
LIN {X 0,Y 298.221,Z 837.779,A -85,B 0,C 180,E1 -17341.296,E2 -17341.296} C_VEL
LIN {X 0,Y 295.628,Z 870.995,A -85,B 0,C 180,E1 -17342.526,E2 -17342.526} C_VEL
LIN {X 0,Y 293.817,Z 885.343,A -85,B 0,C 180,E1 -17343.255,E2 -17343.255} C_VEL
LIN {X 0,Y 291.484,Z 899.17,A -85,B 0,C 180,E1 -17344.276,E2 -17344.276} C_VEL
LIN {X 0,Y 289.487,Z 909.373,A -85,B 0,C 180,E1 -17345.24,E2 -17345.24} C_VEL
LIN {X 0,Y 287.319,Z 919.269,A -85,B 0,C 180,E1 -17346.386,E2 -17346.386} C_VEL
LIN {X 0,Y 285.071,Z 928.84,A -85,B 0,C 180,E1 -17347.723,E2 -17347.723} C_VEL
LIN {X 0,Y 283.297,Z 936.12,A -85,B 0,C 180,E1 -17348.915,E2 -17348.915} C_VEL
LIN {X 0,Y 281.187,Z 944.914,A -85,B 0,C 180,E1 -17350.658,E2 -17350.658} C_VEL
LIN {X 0,Y 279.541,Z 952.371,A -85,B 0,C 180,E1 -17352.438,E2 -17352.438} C_VEL
LIN {X 0,Y 278.194,Z 958.754,A -85,B 0,C 180,E1 -17354.24,E2 -17354.24} C_VEL
LIN {X 0,Y 277.248,Z 964.182,A -85,B 0,C 180,E1 -17356.063,E2 -17356.063} C_VEL
LIN {X 0,Y 276.483,Z 969.486,A -85,B 0,C 180,E1 -17358.265,E2 -17358.265} C_VEL
LIN {X 0,Y 276.299,Z 977.753,A -85,B 0,C 180,E1 -17362.753,E2 -17362.753} C_VEL
LIN {X 0,Y 276.649,Z 981.456,A -85,B 0,C 180,E1 -17365.627,E2 -17365.627} C_VEL
LIN {X 0,Y 276.773,Z 982.689,A -85,B 0,C 180,E1 -17367.087,E2 -17367.087} C_VEL
LIN {X 0,Y 276.911,Z 983.466,A -85,B 0,C 180,E1 -17368.544,E2 -17368.544} C_VEL
LIN {X 0,Y 277.049,Z 983.8,A -85,B 0,C 180,E1 -17369.998,E2 -17369.998} C_VEL
LIN {X 0,Y 276.884,Z 983.677,A -85,B 0,C 180,E1 -17371.452,E2 -17371.452} C_VEL
LIN {X 0,Y 276.722,Z 983.144,A -85,B 0,C 180,E1 -17372.909,E2 -17372.909} C_VEL
LIN {X 0,Y 276.562,Z 982.173,A -85,B 0,C 180,E1 -17374.37,E2 -17374.37} C_VEL
LIN {X 0,Y 276.211,Z 978.901,A -85,B 0,C 180,E1 -17377.307,E2 -17377.307} C_VEL
LIN {X 0,Y 276.135,Z 975.279,A -85,B 0,C 180,E1 -17379.52,E2 -17379.52} C_VEL
LIN {X 0,Y 276.446,Z 970.595,A -85,B 0,C 180,E1 -17381.732,E2 -17381.732} C_VEL
LIN {X 0,Y 277.173,Z 964.736,A -85,B 0,C 180,E1 -17383.936,E2 -17383.936} C_VEL
LIN {X 0,Y 278.084,Z 958.805,A -85,B 0,C 180,E1 -17385.762,E2 -17385.762} C_VEL
LIN {X 0,Y 279.733,Z 950.236,A -85,B 0,C 180,E1 -17387.922,E2 -17387.922} C_VEL
LIN {X 0,Y 281.462,Z 941.531,A -85,B 0,C 180,E1 -17389.697,E2 -17389.697} C_VEL
LIN {X 0,Y 283.626,Z 930.87,A -85,B 0,C 180,E1 -17391.435,E2 -17391.435} C_VEL
LIN {X 0,Y 285.823,Z 918.947,A -85,B 0,C 180,E1 -17392.973,E2 -17392.973} C_VEL
LIN {X 0,Y 287.803,Z 907.091,A -85,B 0,C 180,E1 -17394.141,E2 -17394.141} C_VEL
LIN {X 0,Y 289.642,Z 893.571,A -85,B 0,C 180,E1 -17395.125,E2 -17395.125} C_VEL
LIN {X 0,Y 290.821,Z 880.687,A -85,B 0,C 180,E1 -17395.782,E2 -17395.782} C_VEL
LIN {X 0,Y 291.557,Z 865.109,A -85,B 0,C 180,E1 -17396.256,E2 -17396.256} C_VEL
LIN {X 0,Y 292.428,Z 833.881,A -85,B 0,C 180,E1 -17397.059,E2 -17397.059} C_VEL
LIN {X 0,Y 290.083,Z 805.351,A -85,B 0,C 180,E1 -17398.153,E2 -17398.153} C_VEL
LIN {X 0,Y 287.304,Z 781.677,A -85,B 0,C 180,E1 -17399.189,E2 -17399.189} C_VEL
LIN {X 0,Y 284.557,Z 764.117,A -85,B 0,C 180,E1 -17400.099,E2 -17400.099} C_VEL
LIN {X 0,Y 285.328,Z 759.32,A -85,B 0,C 180,E1 -17401.146,E2 -17401.146} C_VEL
LIN {X 0,Y 286.105,Z 754.508,A -85,B 0,C 180,E1 -17402.292,E2 -17402.292} C_VEL
LIN {X 0,Y 283.737,Z 742.333,A -85,B 0,C 180,E1 -17405.74,E2 -17405.74} C_VEL
LIN {X 0,Y 281.519,Z 732.964,A -85,B 0,C 180,E1 -17408.614,E2 -17408.614} C_VEL
LIN {X 0,Y 278.713,Z 723.066,A -85,B 0,C 180,E1 -17411.938,E2 -17411.938} C_VEL
LIN {X 0,Y 277.253,Z 718.035,A -85,B 0,C 180,E1 -17413.82,E2 -17413.82} C_VEL
LIN {X 0,Y 277.23,Z 717.947,A -85,B 0,C 180,E1 -17417.318,E2 -17417.318} C_VEL
LIN {X 0,Y 277.266,Z 717.947,A -85,B 0,C 180,E1 -17421.788,E2 -17421.788} C_VEL
LIN {X 0,Y 277.294,Z 717.924,A -85,B 0,C 180,E1 -17424.343,E2 -17424.343} C_VEL
LIN {X 0,Y 277.235,Z 717.951,A -85,B 0,C 180,E1 -17427.835,E2 -17427.835} C_VEL
LIN {X 0,Y 277.281,Z 717.942,A -85,B 0,C 180,E1 -17431.212,E2 -17431.212} C_VEL
LIN {X 0,Y 277.305,Z 717.939,A -85,B 0,C 180,E1 -17434.479,E2 -17434.479} C_VEL
LIN {X 0,Y 277.274,Z 717.943,A -85,B 0,C 180,E1 -17437.654,E2 -17437.654} C_VEL
LIN {X 0,Y 277.334,Z 717.938,A -85,B 0,C 180,E1 -17440.766,E2 -17440.766} C_VEL
LIN {X 0,Y 277.423,Z 717.927,A -85,B 0,C 180,E1 -17445.325,E2 -17445.325} C_VEL
LIN {X 0,Y 277.449,Z 717.92,A -85,B 0,C 180,E1 -17449.787,E2 -17449.787} C_VEL
LIN {X 0,Y 277.629,Z 717.902,A -85,B 0,C 180,E1 -17452.729,E2 -17452.729} C_VEL
LIN {X 0,Y 277.81,Z 717.878,A -85,B 0,C 180,E1 -17458.551,E2 -17458.551} C_VEL
LIN {X 0,Y 277.81,Z 717.876,A -85,B 0,C 180,E1 -17461.45,E2 -17461.45} C_VEL
LIN {X 0,Y 277.641,Z 717.898,A -85,B 0,C 180,E1 -17467.271,E2 -17467.271} C_VEL
LIN {X 0,Y 277.496,Z 717.918,A -85,B 0,C 180,E1 -17470.212,E2 -17470.212} C_VEL
LIN {X 0,Y 277.424,Z 717.928,A -85,B 0,C 180,E1 -17474.675,E2 -17474.675} C_VEL
LIN {X 0,Y 277.332,Z 717.934,A -85,B 0,C 180,E1 -17479.235,E2 -17479.235} C_VEL
LIN {X 0,Y 277.282,Z 717.924,A -85,B 0,C 180,E1 -17484.159,E2 -17484.159} C_VEL
LIN {X 0,Y 277.317,Z 717.93,A -85,B 0,C 180,E1 -17487.507,E2 -17487.507} C_VEL
LIN {X 0,Y 277.263,Z 717.951,A -85,B 0,C 180,E1 -17490.483,E2 -17490.483} C_VEL
LIN {X 0,Y 277.291,Z 718.119,A -85,B 0,C 180,E1 -17494.329,E2 -17494.329} C_VEL
LIN {X 0,Y 277.553,Z 719.176,A -85,B 0,C 180,E1 -17494.622,E2 -17494.622} C_VEL
LIN {X 0,Y 279.08,Z 721.848,A -85,B 0,C 180,E1 -17494.954,E2 -17494.954} C_VEL
LIN {X 0,Y 286.816,Z 735.556,A -85,B 0,C 180,E1 -17496.441,E2 -17496.441} C_VEL
LIN {X 0,Y 294.723,Z 751.811,A -85,B 0,C 180,E1 -17497.909,E2 -17497.909} C_VEL
LIN {X 0,Y 294.617,Z 760.173,A -85,B 0,C 180,E1 -17498.143,E2 -17498.143} C_VEL
LIN {X 0,Y 293.774,Z 795.047,A -85,B 0,C 180,E1 -17499.067,E2 -17499.067} C_VEL
LIN {X 0,Y 293.562,Z 809.278,A -85,B 0,C 180,E1 -17499.576,E2 -17499.576} C_VEL
LIN {X 0,Y 293.044,Z 821.484,A -85,B 0,C 180,E1 -17500.285,E2 -17500.285} C_VEL
LIN {X 0,Y 292.034,Z 833.992,A -85,B 0,C 180,E1 -17501.283,E2 -17501.283} C_VEL
LIN {X 0,Y 290.74,Z 845.084,A -85,B 0,C 180,E1 -17502.439,E2 -17502.439} C_VEL
LIN {X 0,Y 289.153,Z 856.251,A -85,B 0,C 180,E1 -17503.945,E2 -17503.945} C_VEL
LIN {X 0,Y 287.535,Z 865.589,A -85,B 0,C 180,E1 -17505.511,E2 -17505.511} C_VEL
LIN {X 0,Y 285.892,Z 873.79,A -85,B 0,C 180,E1 -17507.193,E2 -17507.193} C_VEL
LIN {X 0,Y 284.281,Z 881.249,A -85,B 0,C 180,E1 -17509.073,E2 -17509.073} C_VEL
LIN {X 0,Y 282.912,Z 887.147,A -85,B 0,C 180,E1 -17510.902,E2 -17510.902} C_VEL
LIN {X 0,Y 281.43,Z 893.041,A -85,B 0,C 180,E1 -17513.18,E2 -17513.18} C_VEL
LIN {X 0,Y 279.92,Z 898.33,A -85,B 0,C 180,E1 -17515.95,E2 -17515.95} C_VEL
LIN {X 0,Y 279.142,Z 901.202,A -85,B 0,C 180,E1 -17518.084,E2 -17518.084} C_VEL
LIN {X 0,Y 278.663,Z 902.793,A -85,B 0,C 180,E1 -17519.711,E2 -17519.711} C_VEL
LIN {X 0,Y 278.157,Z 904.181,A -85,B 0,C 180,E1 -17522.169,E2 -17522.169} C_VEL
LIN {X 0,Y 277.847,Z 904.461,A -85,B 0,C 180,E1 -17524.535,E2 -17524.535} C_VEL
LIN {X 0,Y 277.839,Z 904.041,A -85,B 0,C 180,E1 -17526.129,E2 -17526.129} C_VEL
LIN {X 0,Y 277.897,Z 903.198,A -85,B 0,C 180,E1 -17527.709,E2 -17527.709} C_VEL
LIN {X 0,Y 278.071,Z 901.861,A -85,B 0,C 180,E1 -17529.28,E2 -17529.28} C_VEL
LIN {X 0,Y 278.587,Z 898.967,A -85,B 0,C 180,E1 -17531.621,E2 -17531.621} C_VEL
LIN {X 0,Y 279.347,Z 894.95,A -85,B 0,C 180,E1 -17533.936,E2 -17533.936} C_VEL
LIN {X 0,Y 280.282,Z 889.734,A -85,B 0,C 180,E1 -17536.221,E2 -17536.221} C_VEL
LIN {X 0,Y 281.459,Z 883.159,A -85,B 0,C 180,E1 -17538.479,E2 -17538.479} C_VEL
LIN {X 0,Y 282.877,Z 874.886,A -85,B 0,C 180,E1 -17540.709,E2 -17540.709} C_VEL
LIN {X 0,Y 284.268,Z 866.068,A -85,B 0,C 180,E1 -17542.619,E2 -17542.619} C_VEL
LIN {X 0,Y 285.697,Z 856.147,A -85,B 0,C 180,E1 -17544.355,E2 -17544.355} C_VEL
LIN {X 0,Y 286.982,Z 845.908,A -85,B 0,C 180,E1 -17545.789,E2 -17545.789} C_VEL
LIN {X 0,Y 288.14,Z 834.8,A -85,B 0,C 180,E1 -17547.031,E2 -17547.031} C_VEL
LIN {X 0,Y 289.101,Z 822.176,A -85,B 0,C 180,E1 -17548.123,E2 -17548.123} C_VEL
LIN {X 0,Y 289.674,Z 809.045,A -85,B 0,C 180,E1 -17548.934,E2 -17548.934} C_VEL
LIN {X 0,Y 289.922,Z 795.662,A -85,B 0,C 180,E1 -17549.466,E2 -17549.466} C_VEL
LIN {X 0,Y 290.715,Z 748.161,A -85,B 0,C 180,E1 -17550.709,E2 -17550.709} C_VEL
LIN {X 0,Y 285.755,Z 735.759,A -85,B 0,C 180,E1 -17551.504,E2 -17551.504} C_VEL
LIN {X 0,Y 278.371,Z 720.148,A -85,B 0,C 180,E1 -17552.663,E2 -17552.663} C_VEL
LIN {X 0,Y 277.755,Z 718.5,A -85,B 0,C 180,E1 -17552.858,E2 -17552.858} C_VEL
LIN {X 0,Y 277.579,Z 717.935,A -85,B 0,C 180,E1 -17553.268,E2 -17553.268} C_VEL
LIN {X 0,Y 277.604,Z 717.898,A -85,B 0,C 180,E1 -17557.274,E2 -17557.274} C_VEL
LIN {X 0,Y 277.459,Z 717.915,A -85,B 0,C 180,E1 -17560.215,E2 -17560.215} C_VEL
LIN {X 0,Y 277.414,Z 717.916,A -85,B 0,C 180,E1 -17564.677,E2 -17564.677} C_VEL
LIN {X 0,Y 277.288,Z 717.929,A -85,B 0,C 180,E1 -17569.24,E2 -17569.24} C_VEL
LIN {X 0,Y 277.266,Z 717.946,A -85,B 0,C 180,E1 -17573.928,E2 -17573.928} C_VEL
LIN {X 0,Y 277.241,Z 717.929,A -85,B 0,C 180,E1 -17577.47,E2 -17577.47} C_VEL
LIN {X 0,Y 277.234,Z 717.951,A -85,B 0,C 180,E1 -17580.467,E2 -17580.467} C_VEL
LIN {X 0,Y 277.252,Z 717.919,A -85,B 0,C 180,E1 -17583.897,E2 -17583.897} C_VEL
LIN {X 0,Y 277.257,Z 717.935,A -85,B 0,C 180,E1 -17587.473,E2 -17587.473} C_VEL
LIN {X 0,Y 277.187,Z 717.958,A -85,B 0,C 180,E1 -17591.243,E2 -17591.243} C_VEL
LIN {X 0,Y 277.181,Z 717.959,A -85,B 0,C 180,E1 -17595.233,E2 -17595.233} C_VEL
LIN {X 0,Y 277.191,Z 717.956,A -85,B 0,C 180,E1 -17598.759,E2 -17598.759} C_VEL
LIN {X 0,Y 277.298,Z 718.137,A -85,B 0,C 180,E1 -17602.101,E2 -17602.101} C_VEL
LIN {X 0,Y 277.517,Z 719,A -85,B 0,C 180,E1 -17602.319,E2 -17602.319} C_VEL
LIN {X 0,Y 286.044,Z 743.212,A -85,B 0,C 180,E1 -17603.693,E2 -17603.693} C_VEL
LIN {X 0,Y 284.548,Z 796.707,A -85,B 0,C 180,E1 -17605.491,E2 -17605.491} C_VEL
LIN {X 0,Y 284.198,Z 808.261,A -85,B 0,C 180,E1 -17606.085,E2 -17606.085} C_VEL
LIN {X 0,Y 283.781,Z 818.287,A -85,B 0,C 180,E1 -17606.774,E2 -17606.774} C_VEL
LIN {X 0,Y 283.116,Z 828.713,A -85,B 0,C 180,E1 -17607.677,E2 -17607.677} C_VEL
LIN {X 0,Y 282.448,Z 838.332,A -85,B 0,C 180,E1 -17608.706,E2 -17608.706} C_VEL
LIN {X 0,Y 281.695,Z 847.315,A -85,B 0,C 180,E1 -17609.861,E2 -17609.861} C_VEL
LIN {X 0,Y 280.938,Z 856.264,A -85,B 0,C 180,E1 -17611.237,E2 -17611.237} C_VEL
LIN {X 0,Y 279.814,Z 860.873,A -85,B 0,C 180,E1 -17612,E2 -17612} C_VEL
LIN {X 0,Y 276.299,Z 867.793,A -85,B 0,C 180,E1 -17613.264,E2 -17613.264} C_VEL
LIN {X 0,Y 273.43,Z 873.036,A -85,B 0,C 180,E1 -17614.349,E2 -17614.349} C_VEL
LIN {X 0,Y 272.054,Z 876.857,A -85,B 0,C 180,E1 -17615.247,E2 -17615.247} C_VEL
LIN {X 0,Y 271.858,Z 878.087,A -85,B 0,C 180,E1 -17615.563,E2 -17615.563} C_VEL
LIN {X 0,Y 271.238,Z 885.765,A -85,B 0,C 180,E1 -17617.932,E2 -17617.932} C_VEL
LIN {X 0,Y 270.89,Z 890.401,A -85,B 0,C 180,E1 -17619.639,E2 -17619.639} C_VEL
LIN {X 0,Y 270.577,Z 895.204,A -85,B 0,C 180,E1 -17621.839,E2 -17621.839} C_VEL
LIN {X 0,Y 270.477,Z 898.899,A -85,B 0,C 180,E1 -17624.035,E2 -17624.035} C_VEL
LIN {X 0,Y 270.574,Z 901.825,A -85,B 0,C 180,E1 -17626.481,E2 -17626.481} C_VEL
LIN {X 0,Y 270.819,Z 903.164,A -85,B 0,C 180,E1 -17628.018,E2 -17628.018} C_VEL
LIN {X 0,Y 271.25,Z 904.077,A -85,B 0,C 180,E1 -17629.931,E2 -17629.931} C_VEL
LIN {X 0,Y 272.068,Z 904.221,A -85,B 0,C 180,E1 -17632.579,E2 -17632.579} C_VEL
LIN {X 0,Y 273.47,Z 902.607,A -85,B 0,C 180,E1 -17635.578,E2 -17635.578} C_VEL
LIN {X 0,Y 274.431,Z 901.112,A -85,B 0,C 180,E1 -17637.186,E2 -17637.186} C_VEL
LIN {X 0,Y 275.777,Z 898.292,A -85,B 0,C 180,E1 -17639.27,E2 -17639.27} C_VEL
LIN {X 0,Y 277.504,Z 894.163,A -85,B 0,C 180,E1 -17641.451,E2 -17641.451} C_VEL
LIN {X 0,Y 279.556,Z 888.749,A -85,B 0,C 180,E1 -17643.603,E2 -17643.603} C_VEL
LIN {X 0,Y 281.446,Z 883.254,A -85,B 0,C 180,E1 -17645.373,E2 -17645.373} C_VEL
LIN {X 0,Y 283.463,Z 876.643,A -85,B 0,C 180,E1 -17647.121,E2 -17647.121} C_VEL
LIN {X 0,Y 285.534,Z 869.177,A -85,B 0,C 180,E1 -17648.733,E2 -17648.733} C_VEL
LIN {X 0,Y 287.51,Z 860.933,A -85,B 0,C 180,E1 -17650.208,E2 -17650.208} C_VEL
LIN {X 0,Y 289.433,Z 851.851,A -85,B 0,C 180,E1 -17651.556,E2 -17651.556} C_VEL
LIN {X 0,Y 290.923,Z 843.764,A -85,B 0,C 180,E1 -17652.557,E2 -17652.557} C_VEL
LIN {X 0,Y 292.375,Z 834.065,A -85,B 0,C 180,E1 -17653.554,E2 -17653.554} C_VEL
LIN {X 0,Y 293.492,Z 824.149,A -85,B 0,C 180,E1 -17654.385,E2 -17654.385} C_VEL
LIN {X 0,Y 294.405,Z 813.869,A -85,B 0,C 180,E1 -17655.047,E2 -17655.047} C_VEL
LIN {X 0,Y 295.379,Z 796.861,A -85,B 0,C 180,E1 -17655.864,E2 -17655.864} C_VEL
LIN {X 0,Y 297.609,Z 769.834,A -85,B 0,C 180,E1 -17656.911,E2 -17656.911} C_VEL
LIN {X 0,Y 298.257,Z 761.112,A -85,B 0,C 180,E1 -17657.265,E2 -17657.265} C_VEL
LIN {X 0,Y 294.339,Z 753.447,A -85,B 0,C 180,E1 -17658.648,E2 -17658.648} C_VEL
LIN {X 0,Y 289.917,Z 746.11,A -85,B 0,C 180,E1 -17660.314,E2 -17660.314} C_VEL
LIN {X 0,Y 287.503,Z 742.349,A -85,B 0,C 180,E1 -17661.315,E2 -17661.315} C_VEL
LIN {X 0,Y 285.491,Z 739.308,A -85,B 0,C 180,E1 -17662.218,E2 -17662.218} C_VEL
LIN {X 0,Y 283.062,Z 735.904,A -85,B 0,C 180,E1 -17663.361,E2 -17663.361} C_VEL
LIN {X 0,Y 282.253,Z 734.795,A -85,B 0,C 180,E1 -17663.781,E2 -17663.781} C_VEL
LIN {X 0,Y 279.731,Z 731.511,A -85,B 0,C 180,E1 -17665.144,E2 -17665.144} C_VEL
LIN {X 0,Y 279.091,Z 730.109,A -85,B 0,C 180,E1 -17665.596,E2 -17665.596} C_VEL
LIN {X 0,Y 276.505,Z 727.848,A -85,B 0,C 180,E1 -17667.173,E2 -17667.173} C_VEL
LIN {X 0,Y 274.762,Z 724.668,A -85,B 0,C 180,E1 -17668.659,E2 -17668.659} C_VEL
LIN {X 0,Y 271.604,Z 722.283,A -85,B 0,C 180,E1 -17671.677,E2 -17671.677} C_VEL
LIN {X 0,Y 270.54,Z 720.225,A -85,B 0,C 180,E1 -17673.766,E2 -17673.766} C_VEL
LIN {X 0,Y 270.588,Z 720.331,A -85,B 0,C 180,E1 -17676.683,E2 -17676.683} C_VEL
LIN {X 0,Y 271.542,Z 722.172,A -85,B 0,C 180,E1 -17680.319,E2 -17680.319} C_VEL
LIN {X 0,Y 272.605,Z 723.383,A -85,B 0,C 180,E1 -17682.09,E2 -17682.09} C_VEL
LIN {X 0,Y 274.027,Z 725.6,A -85,B 0,C 180,E1 -17684.098,E2 -17684.098} C_VEL
LIN {X 0,Y 276.579,Z 729.159,A -85,B 0,C 180,E1 -17686.677,E2 -17686.677} C_VEL
LIN {X 0,Y 279.501,Z 734.321,A -85,B 0,C 180,E1 -17689.171,E2 -17689.171} C_VEL
LIN {X 0,Y 280.856,Z 739.199,A -85,B 0,C 180,E1 -17690.463,E2 -17690.463} C_VEL
LIN {X 0,Y 283.924,Z 748.207,A -85,B 0,C 180,E1 -17692.382,E2 -17692.382} C_VEL
LIN {X 0,Y 288.4,Z 761.033,A -85,B 0,C 180,E1 -17694.722,E2 -17694.722} C_VEL
LIN {X 0,Y 289.45,Z 764.932,A -85,B 0,C 180,E1 -17695.268,E2 -17695.268} C_VEL
LIN {X 0,Y 291.258,Z 785.302,A -85,B 0,C 180,E1 -17697.029,E2 -17697.029} C_VEL
LIN {X 0,Y 292.539,Z 807.358,A -85,B 0,C 180,E1 -17698.623,E2 -17698.623} C_VEL
LIN {X 0,Y 292.891,Z 818.669,A -85,B 0,C 180,E1 -17699.317,E2 -17699.317} C_VEL
LIN {X 0,Y 292.921,Z 838.922,A -85,B 0,C 180,E1 -17700.406,E2 -17700.406} C_VEL
LIN {X 0,Y 290.292,Z 869.856,A -85,B 0,C 180,E1 -17701.581,E2 -17701.581} C_VEL
LIN {X 0,Y 288.398,Z 883.956,A -85,B 0,C 180,E1 -17702.318,E2 -17702.318} C_VEL
LIN {X 0,Y 285.942,Z 897.622,A -85,B 0,C 180,E1 -17703.347,E2 -17703.347} C_VEL
LIN {X 0,Y 283.842,Z 907.776,A -85,B 0,C 180,E1 -17704.32,E2 -17704.32} C_VEL
LIN {X 0,Y 281.519,Z 917.735,A -85,B 0,C 180,E1 -17705.476,E2 -17705.476} C_VEL
LIN {X 0,Y 279.359,Z 926.229,A -85,B 0,C 180,E1 -17706.655,E2 -17706.655} C_VEL
LIN {X 0,Y 277.206,Z 934.552,A -85,B 0,C 180,E1 -17708.038,E2 -17708.038} C_VEL
LIN {X 0,Y 274.931,Z 943.354,A -85,B 0,C 180,E1 -17709.81,E2 -17709.81} C_VEL
LIN {X 0,Y 273.042,Z 950.856,A -85,B 0,C 180,E1 -17711.618,E2 -17711.618} C_VEL
LIN {X 0,Y 271.46,Z 957.24,A -85,B 0,C 180,E1 -17713.452,E2 -17713.452} C_VEL
LIN {X 0,Y 270.273,Z 963.602,A -85,B 0,C 180,E1 -17715.696,E2 -17715.696} C_VEL
LIN {X 0,Y 269.458,Z 968.777,A -85,B 0,C 180,E1 -17717.954,E2 -17717.954} C_VEL
LIN {X 0,Y 269.18,Z 972.892,A -85,B 0,C 180,E1 -17720.227,E2 -17720.227} C_VEL
LIN {X 0,Y 269.236,Z 976.873,A -85,B 0,C 180,E1 -17722.717,E2 -17722.717} C_VEL
LIN {X 0,Y 269.567,Z 980.377,A -85,B 0,C 180,E1 -17725.512,E2 -17725.512} C_VEL
LIN {X 0,Y 269.723,Z 981.63,A -85,B 0,C 180,E1 -17727.011,E2 -17727.011} C_VEL
LIN {X 0,Y 269.871,Z 982.435,A -85,B 0,C 180,E1 -17728.506,E2 -17728.506} C_VEL
LIN {X 0,Y 270.017,Z 982.782,A -85,B 0,C 180,E1 -17729.998,E2 -17729.998} C_VEL
LIN {X 0,Y 269.841,Z 982.668,A -85,B 0,C 180,E1 -17731.49,E2 -17731.49} C_VEL
LIN {X 0,Y 269.664,Z 982.143,A -85,B 0,C 180,E1 -17732.986,E2 -17732.986} C_VEL
LIN {X 0,Y 269.486,Z 981.192,A -85,B 0,C 180,E1 -17734.485,E2 -17734.485} C_VEL
LIN {X 0,Y 269.158,Z 978.409,A -85,B 0,C 180,E1 -17737.152,E2 -17737.152} C_VEL
LIN {X 0,Y 269.089,Z 974.356,A -85,B 0,C 180,E1 -17739.772,E2 -17739.772} C_VEL
LIN {X 0,Y 269.437,Z 969.706,A -85,B 0,C 180,E1 -17742.042,E2 -17742.042} C_VEL
LIN {X 0,Y 270.397,Z 962.81,A -85,B 0,C 180,E1 -17744.677,E2 -17744.677} C_VEL
LIN {X 0,Y 271.633,Z 955.778,A -85,B 0,C 180,E1 -17746.802,E2 -17746.802} C_VEL
LIN {X 0,Y 273.576,Z 946.177,A -85,B 0,C 180,E1 -17749.117,E2 -17749.117} C_VEL
LIN {X 0,Y 275.61,Z 936.862,A -85,B 0,C 180,E1 -17750.913,E2 -17750.913} C_VEL
LIN {X 0,Y 277.728,Z 926.652,A -85,B 0,C 180,E1 -17752.501,E2 -17752.501} C_VEL
LIN {X 0,Y 279.897,Z 915.398,A -85,B 0,C 180,E1 -17753.881,E2 -17753.881} C_VEL
LIN {X 0,Y 281.97,Z 902.868,A -85,B 0,C 180,E1 -17755.067,E2 -17755.067} C_VEL
LIN {X 0,Y 283.655,Z 890.268,A -85,B 0,C 180,E1 -17755.939,E2 -17755.939} C_VEL
LIN {X 0,Y 284.776,Z 877.594,A -85,B 0,C 180,E1 -17756.548,E2 -17756.548} C_VEL
LIN {X 0,Y 285.609,Z 857.383,A -85,B 0,C 180,E1 -17757.13,E2 -17757.13} C_VEL
LIN {X 0,Y 286.2,Z 833.685,A -85,B 0,C 180,E1 -17757.763,E2 -17757.763} C_VEL
LIN {X 0,Y 283.923,Z 805.97,A -85,B 0,C 180,E1 -17758.865,E2 -17758.865} C_VEL
LIN {X 0,Y 281.13,Z 781.901,A -85,B 0,C 180,E1 -17759.953,E2 -17759.953} C_VEL
LIN {X 0,Y 278.173,Z 762.724,A -85,B 0,C 180,E1 -17761.008,E2 -17761.008} C_VEL
LIN {X 0,Y 279.252,Z 757.048,A -85,B 0,C 180,E1 -17762.328,E2 -17762.328} C_VEL
LIN {X 0,Y 278.589,Z 752.091,A -85,B 0,C 180,E1 -17763.708,E2 -17763.708} C_VEL
LIN {X 0,Y 276.435,Z 741.786,A -85,B 0,C 180,E1 -17766.79,E2 -17766.79} C_VEL
LIN {X 0,Y 274.115,Z 732.296,A -85,B 0,C 180,E1 -17769.861,E2 -17769.861} C_VEL
LIN {X 0,Y 271.134,Z 722.233,A -85,B 0,C 180,E1 -17773.466,E2 -17773.466} C_VEL
LIN {X 0,Y 270.192,Z 718.916,A -85,B 0,C 180,E1 -17774.8,E2 -17774.8} C_VEL
LIN {X 0,Y 270.198,Z 718.818,A -85,B 0,C 180,E1 -17778.961,E2 -17778.961} C_VEL
LIN {X 0,Y 270.229,Z 718.814,A -85,B 0,C 180,E1 -17783.261,E2 -17783.261} C_VEL
LIN {X 0,Y 270.195,Z 718.828,A -85,B 0,C 180,E1 -17786.891,E2 -17786.891} C_VEL
LIN {X 0,Y 270.219,Z 718.826,A -85,B 0,C 180,E1 -17790.386,E2 -17790.386} C_VEL
LIN {X 0,Y 270.255,Z 718.82,A -85,B 0,C 180,E1 -17793.763,E2 -17793.763} C_VEL
LIN {X 0,Y 270.223,Z 718.826,A -85,B 0,C 180,E1 -17797.038,E2 -17797.038} C_VEL
LIN {X 0,Y 270.291,Z 718.817,A -85,B 0,C 180,E1 -17800.244,E2 -17800.244} C_VEL
LIN {X 0,Y 270.392,Z 718.803,A -85,B 0,C 180,E1 -17804.935,E2 -17804.935} C_VEL
LIN {X 0,Y 270.401,Z 718.802,A -85,B 0,C 180,E1 -17809.518,E2 -17809.518} C_VEL
LIN {X 0,Y 270.587,Z 718.775,A -85,B 0,C 180,E1 -17812.538,E2 -17812.538} C_VEL
LIN {X 0,Y 270.776,Z 718.754,A -85,B 0,C 180,E1 -17818.513,E2 -17818.513} C_VEL
LIN {X 0,Y 270.776,Z 718.752,A -85,B 0,C 180,E1 -17821.488,E2 -17821.488} C_VEL
LIN {X 0,Y 270.599,Z 718.775,A -85,B 0,C 180,E1 -17827.462,E2 -17827.462} C_VEL
LIN {X 0,Y 270.431,Z 718.8,A -85,B 0,C 180,E1 -17830.482,E2 -17830.482} C_VEL
LIN {X 0,Y 270.392,Z 718.8,A -85,B 0,C 180,E1 -17835.066,E2 -17835.066} C_VEL
LIN {X 0,Y 270.289,Z 718.812,A -85,B 0,C 180,E1 -17839.757,E2 -17839.757} C_VEL
LIN {X 0,Y 270.228,Z 718.805,A -85,B 0,C 180,E1 -17844.59,E2 -17844.59} C_VEL
LIN {X 0,Y 270.261,Z 718.805,A -85,B 0,C 180,E1 -17847.91,E2 -17847.91} C_VEL
LIN {X 0,Y 270.175,Z 718.828,A -85,B 0,C 180,E1 -17851.35,E2 -17851.35} C_VEL
LIN {X 0,Y 270.255,Z 719.052,A -85,B 0,C 180,E1 -17853.314,E2 -17853.314} C_VEL
LIN {X 0,Y 270.487,Z 720.041,A -85,B 0,C 180,E1 -17853.58,E2 -17853.58} C_VEL
LIN {X 0,Y 271.974,Z 722.68,A -85,B 0,C 180,E1 -17853.922,E2 -17853.922} C_VEL
LIN {X 0,Y 278.995,Z 734.599,A -85,B 0,C 180,E1 -17855.352,E2 -17855.352} C_VEL
LIN {X 0,Y 286.359,Z 749.076,A -85,B 0,C 180,E1 -17856.798,E2 -17856.798} C_VEL
LIN {X 0,Y 288.737,Z 754.125,A -85,B 0,C 180,E1 -17857.251,E2 -17857.251} C_VEL
LIN {X 0,Y 287.644,Z 795.668,A -85,B 0,C 180,E1 -17858.373,E2 -17858.373} C_VEL
LIN {X 0,Y 287.425,Z 810.138,A -85,B 0,C 180,E1 -17858.899,E2 -17858.899} C_VEL
LIN {X 0,Y 286.938,Z 821.449,A -85,B 0,C 180,E1 -17859.556,E2 -17859.556} C_VEL
LIN {X 0,Y 285.943,Z 833.422,A -85,B 0,C 180,E1 -17860.503,E2 -17860.503} C_VEL
LIN {X 0,Y 284.627,Z 844.541,A -85,B 0,C 180,E1 -17861.649,E2 -17861.649} C_VEL
LIN {X 0,Y 282.99,Z 855.923,A -85,B 0,C 180,E1 -17863.157,E2 -17863.157} C_VEL
LIN {X 0,Y 281.282,Z 865.49,A -85,B 0,C 180,E1 -17864.756,E2 -17864.756} C_VEL
LIN {X 0,Y 279.355,Z 874.787,A -85,B 0,C 180,E1 -17866.681,E2 -17866.681} C_VEL
LIN {X 0,Y 277.464,Z 883.003,A -85,B 0,C 180,E1 -17868.813,E2 -17868.813} C_VEL
LIN {X 0,Y 275.903,Z 889.407,A -85,B 0,C 180,E1 -17870.92,E2 -17870.92} C_VEL
LIN {X 0,Y 274.418,Z 894.764,A -85,B 0,C 180,E1 -17873.138,E2 -17873.138} C_VEL
LIN {X 0,Y 273.109,Z 899.163,A -85,B 0,C 180,E1 -17875.522,E2 -17875.522} C_VEL
LIN {X 0,Y 272.448,Z 901.524,A -85,B 0,C 180,E1 -17877.203,E2 -17877.203} C_VEL
LIN {X 0,Y 271.873,Z 903.267,A -85,B 0,C 180,E1 -17878.871,E2 -17878.871} C_VEL
LIN {X 0,Y 271.196,Z 905.119,A -85,B 0,C 180,E1 -17881.777,E2 -17881.777} C_VEL
LIN {X 0,Y 270.887,Z 905.493,A -85,B 0,C 180,E1 -17883.832,E2 -17883.832} C_VEL
LIN {X 0,Y 270.803,Z 905.292,A -85,B 0,C 180,E1 -17885.468,E2 -17885.468} C_VEL
LIN {X 0,Y 270.844,Z 904.576,A -85,B 0,C 180,E1 -17887.096,E2 -17887.096} C_VEL
LIN {X 0,Y 271.02,Z 903.195,A -85,B 0,C 180,E1 -17888.995,E2 -17888.995} C_VEL
LIN {X 0,Y 271.412,Z 900.823,A -85,B 0,C 180,E1 -17891.117,E2 -17891.117} C_VEL
LIN {X 0,Y 272.171,Z 897.099,A -85,B 0,C 180,E1 -17893.501,E2 -17893.501} C_VEL
LIN {X 0,Y 273.056,Z 892.204,A -85,B 0,C 180,E1 -17895.849,E2 -17895.849} C_VEL
LIN {X 0,Y 274.239,Z 885.942,A -85,B 0,C 180,E1 -17898.172,E2 -17898.172} C_VEL
LIN {X 0,Y 275.654,Z 878.146,A -85,B 0,C 180,E1 -17900.463,E2 -17900.463} C_VEL
LIN {X 0,Y 277.11,Z 869.438,A -85,B 0,C 180,E1 -17902.51,E2 -17902.51} C_VEL
LIN {X 0,Y 278.657,Z 859.378,A -85,B 0,C 180,E1 -17904.394,E2 -17904.394} C_VEL
LIN {X 0,Y 280.142,Z 848.355,A -85,B 0,C 180,E1 -17906.046,E2 -17906.046} C_VEL
LIN {X 0,Y 281.417,Z 836.982,A -85,B 0,C 180,E1 -17907.38,E2 -17907.38} C_VEL
LIN {X 0,Y 282.39,Z 825.059,A -85,B 0,C 180,E1 -17908.467,E2 -17908.467} C_VEL
LIN {X 0,Y 283.029,Z 812.545,A -85,B 0,C 180,E1 -17909.317,E2 -17909.317} C_VEL
LIN {X 0,Y 283.354,Z 799.29,A -85,B 0,C 180,E1 -17909.908,E2 -17909.908} C_VEL
LIN {X 0,Y 284.127,Z 757.284,A -85,B 0,C 180,E1 -17911.042,E2 -17911.042} C_VEL
LIN {X 0,Y 284.131,Z 749.511,A -85,B 0,C 180,E1 -17911.262,E2 -17911.262} C_VEL
LIN {X 0,Y 278.676,Z 736.349,A -85,B 0,C 180,E1 -17912.156,E2 -17912.156} C_VEL
LIN {X 0,Y 272.013,Z 722.324,A -85,B 0,C 180,E1 -17913.239,E2 -17913.239} C_VEL
LIN {X 0,Y 270.613,Z 719.493,A -85,B 0,C 180,E1 -17913.539,E2 -17913.539} C_VEL
LIN {X 0,Y 270.463,Z 718.83,A -85,B 0,C 180,E1 -17913.913,E2 -17913.913} C_VEL
LIN {X 0,Y 270.566,Z 718.775,A -85,B 0,C 180,E1 -17917.465,E2 -17917.465} C_VEL
LIN {X 0,Y 270.393,Z 718.794,A -85,B 0,C 180,E1 -17920.485,E2 -17920.485} C_VEL
LIN {X 0,Y 270.373,Z 718.793,A -85,B 0,C 180,E1 -17925.069,E2 -17925.069} C_VEL
LIN {X 0,Y 270.228,Z 718.805,A -85,B 0,C 180,E1 -17929.763,E2 -17929.763} C_VEL
LIN {X 0,Y 270.19,Z 718.822,A -85,B 0,C 180,E1 -17934.439,E2 -17934.439} C_VEL
LIN {X 0,Y 270.19,Z 718.812,A -85,B 0,C 180,E1 -17937.92,E2 -17937.92} C_VEL
LIN {X 0,Y 270.175,Z 718.828,A -85,B 0,C 180,E1 -17941.352,E2 -17941.352} C_VEL
LIN {X 0,Y 270.204,Z 718.791,A -85,B 0,C 180,E1 -17944.908,E2 -17944.908} C_VEL
LIN {X 0,Y 270.205,Z 718.823,A -85,B 0,C 180,E1 -17948.712,E2 -17948.712} C_VEL
LIN {X 0,Y 270.153,Z 718.834,A -85,B 0,C 180,E1 -17953.245,E2 -17953.245} C_VEL
LIN {X 0,Y 270.158,Z 718.833,A -85,B 0,C 180,E1 -17957.438,E2 -17957.438} C_VEL
LIN {X 0,Y 270.253,Z 719.044,A -85,B 0,C 180,E1 -17961.695,E2 -17961.695} C_VEL
LIN {X 0,Y 270.574,Z 720.255,A -85,B 0,C 180,E1 -17961.94,E2 -17961.94} C_VEL
LIN {X 0,Y 279.157,Z 744.615,A -85,B 0,C 180,E1 -17963.357,E2 -17963.357} C_VEL
LIN {X 0,Y 277.587,Z 797.887,A -85,B 0,C 180,E1 -17965.218,E2 -17965.218} C_VEL
LIN {X 0,Y 277.274,Z 808.571,A -85,B 0,C 180,E1 -17965.779,E2 -17965.779} C_VEL
LIN {X 0,Y 276.853,Z 818.889,A -85,B 0,C 180,E1 -17966.501,E2 -17966.501} C_VEL
LIN {X 0,Y 276.114,Z 829.658,A -85,B 0,C 180,E1 -17967.455,E2 -17967.455} C_VEL
LIN {X 0,Y 275.466,Z 838.912,A -85,B 0,C 180,E1 -17968.465,E2 -17968.465} C_VEL
LIN {X 0,Y 274.705,Z 847.922,A -85,B 0,C 180,E1 -17969.64,E2 -17969.64} C_VEL
LIN {X 0,Y 273.928,Z 856.868,A -85,B 0,C 180,E1 -17971.035,E2 -17971.035} C_VEL
LIN {X 0,Y 273.243,Z 864.446,A -85,B 0,C 180,E1 -17972.42,E2 -17972.42} C_VEL
LIN {X 0,Y 272.521,Z 871.808,A -85,B 0,C 180,E1 -17973.997,E2 -17973.997} C_VEL
LIN {X 0,Y 271.858,Z 878.087,A -85,B 0,C 180,E1 -17975.563,E2 -17975.563} C_VEL
LIN {X 0,Y 270.878,Z 881.701,A -85,B 0,C 180,E1 -17976.527,E2 -17976.527} C_VEL
LIN {X 0,Y 267.589,Z 887.04,A -85,B 0,C 180,E1 -17978.162,E2 -17978.162} C_VEL
LIN {X 0,Y 264.404,Z 891.85,A -85,B 0,C 180,E1 -17979.919,E2 -17979.919} C_VEL
LIN {X 0,Y 263.602,Z 894.43,A -85,B 0,C 180,E1 -17981.058,E2 -17981.058} C_VEL
LIN {X 0,Y 263.442,Z 899.459,A -85,B 0,C 180,E1 -17983.827,E2 -17983.827} C_VEL
LIN {X 0,Y 263.504,Z 902.399,A -85,B 0,C 180,E1 -17986.111,E2 -17986.111} C_VEL
LIN {X 0,Y 264.046,Z 904.852,A -85,B 0,C 180,E1 -17989.262,E2 -17989.262} C_VEL
LIN {X 0,Y 264.476,Z 905.392,A -85,B 0,C 180,E1 -17990.825,E2 -17990.825} C_VEL
LIN {X 0,Y 264.987,Z 905.489,A -85,B 0,C 180,E1 -17992.379,E2 -17992.379} C_VEL
LIN {X 0,Y 266.436,Z 904.375,A -85,B 0,C 180,E1 -17995.461,E2 -17995.461} C_VEL
LIN {X 0,Y 267.415,Z 903.021,A -85,B 0,C 180,E1 -17997.098,E2 -17997.098} C_VEL
LIN {X 0,Y 269.374,Z 899.33,A -85,B 0,C 180,E1 -18000,E2 -18000} C_VEL
LIN {X 0,Y 271.275,Z 895.172,A -85,B 0,C 180,E1 -18002.227,E2 -18002.227} C_VEL
LIN {X 0,Y 273.134,Z 890.798,A -85,B 0,C 180,E1 -18004.057,E2 -18004.057} C_VEL
LIN {X 0,Y 275.509,Z 884.226,A -85,B 0,C 180,E1 -18006.224,E2 -18006.224} C_VEL
LIN {X 0,Y 277.606,Z 877.845,A -85,B 0,C 180,E1 -18007.923,E2 -18007.923} C_VEL
LIN {X 0,Y 279.599,Z 871.235,A -85,B 0,C 180,E1 -18009.403,E2 -18009.403} C_VEL
LIN {X 0,Y 281.799,Z 862.865,A -85,B 0,C 180,E1 -18010.962,E2 -18010.962} C_VEL
LIN {X 0,Y 283.6,Z 855.154,A -85,B 0,C 180,E1 -18012.16,E2 -18012.16} C_VEL
LIN {X 0,Y 285.415,Z 845.966,A -85,B 0,C 180,E1 -18013.347,E2 -18013.347} C_VEL
LIN {X 0,Y 286.975,Z 836.493,A -85,B 0,C 180,E1 -18014.357,E2 -18014.357} C_VEL
LIN {X 0,Y 288.313,Z 825.924,A -85,B 0,C 180,E1 -18015.282,E2 -18015.282} C_VEL
LIN {X 0,Y 289.31,Z 815.981,A -85,B 0,C 180,E1 -18015.95,E2 -18015.95} C_VEL
LIN {X 0,Y 290.273,Z 801.783,A -85,B 0,C 180,E1 -18016.664,E2 -18016.664} C_VEL
LIN {X 0,Y 292.399,Z 775.162,A -85,B 0,C 180,E1 -18017.757,E2 -18017.757} C_VEL
LIN {X 0,Y 293.385,Z 764.146,A -85,B 0,C 180,E1 -18018.209,E2 -18018.209} C_VEL
LIN {X 0,Y 289.11,Z 755.855,A -85,B 0,C 180,E1 -18019.852,E2 -18019.852} C_VEL
LIN {X 0,Y 284.421,Z 748.158,A -85,B 0,C 180,E1 -18021.848,E2 -18021.848} C_VEL
LIN {X 0,Y 282.243,Z 744.92,A -85,B 0,C 180,E1 -18022.876,E2 -18022.876} C_VEL
LIN {X 0,Y 279.629,Z 741.004,A -85,B 0,C 180,E1 -18024.254,E2 -18024.254} C_VEL
LIN {X 0,Y 277.189,Z 737.579,A -85,B 0,C 180,E1 -18025.684,E2 -18025.684} C_VEL
LIN {X 0,Y 276.573,Z 736.528,A -85,B 0,C 180,E1 -18026.1,E2 -18026.1} C_VEL
LIN {X 0,Y 274.137,Z 734.008,A -85,B 0,C 180,E1 -18027.74,E2 -18027.74} C_VEL
LIN {X 0,Y 272.911,Z 731.465,A -85,B 0,C 180,E1 -18028.884,E2 -18028.884} C_VEL
LIN {X 0,Y 269.808,Z 728.936,A -85,B 0,C 180,E1 -18032.055,E2 -18032.055} C_VEL
LIN {X 0,Y 268.769,Z 727.011,A -85,B 0,C 180,E1 -18034.212,E2 -18034.212} C_VEL
LIN {X 0,Y 268.011,Z 727.086,A -85,B 0,C 180,E1 -18037.094,E2 -18037.094} C_VEL
LIN {X 0,Y 268.645,Z 728.803,A -85,B 0,C 180,E1 -18040.65,E2 -18040.65} C_VEL
LIN {X 0,Y 269.982,Z 730.637,A -85,B 0,C 180,E1 -18042.883,E2 -18042.883} C_VEL
LIN {X 0,Y 271.37,Z 732.962,A -85,B 0,C 180,E1 -18044.589,E2 -18044.589} C_VEL
LIN {X 0,Y 273.888,Z 736.084,A -85,B 0,C 180,E1 -18046.755,E2 -18046.755} C_VEL
LIN {X 0,Y 276.455,Z 740.203,A -85,B 0,C 180,E1 -18048.624,E2 -18048.624} C_VEL
LIN {X 0,Y 279.499,Z 749.572,A -85,B 0,C 180,E1 -18050.885,E2 -18050.885} C_VEL
LIN {X 0,Y 284.512,Z 765.235,A -85,B 0,C 180,E1 -18053.88,E2 -18053.88} C_VEL
LIN {X 0,Y 285.262,Z 768.422,A -85,B 0,C 180,E1 -18054.338,E2 -18054.338} C_VEL
LIN {X 0,Y 286.712,Z 787.622,A -85,B 0,C 180,E1 -18056.056,E2 -18056.056} C_VEL
LIN {X 0,Y 287.716,Z 809.36,A -85,B 0,C 180,E1 -18057.673,E2 -18057.673} C_VEL
LIN {X 0,Y 287.909,Z 820.488,A -85,B 0,C 180,E1 -18058.381,E2 -18058.381} C_VEL
LIN {X 0,Y 287.753,Z 840.162,A -85,B 0,C 180,E1 -18059.468,E2 -18059.468} C_VEL
LIN {X 0,Y 285.195,Z 868.279,A -85,B 0,C 180,E1 -18060.571,E2 -18060.571} C_VEL
LIN {X 0,Y 283.084,Z 882.806,A -85,B 0,C 180,E1 -18061.348,E2 -18061.348} C_VEL
LIN {X 0,Y 280.488,Z 896.344,A -85,B 0,C 180,E1 -18062.382,E2 -18062.382} C_VEL
LIN {X 0,Y 278.278,Z 906.465,A -85,B 0,C 180,E1 -18063.364,E2 -18063.364} C_VEL
LIN {X 0,Y 275.762,Z 916.343,A -85,B 0,C 180,E1 -18064.526,E2 -18064.526} C_VEL
LIN {X 0,Y 273.178,Z 925.831,A -85,B 0,C 180,E1 -18065.893,E2 -18065.893} C_VEL
LIN {X 0,Y 270.648,Z 934.927,A -85,B 0,C 180,E1 -18067.477,E2 -18067.477} C_VEL
LIN {X 0,Y 268.736,Z 941.917,A -85,B 0,C 180,E1 -18068.923,E2 -18068.923} C_VEL
LIN {X 0,Y 266.629,Z 949.394,A -85,B 0,C 180,E1 -18070.76,E2 -18070.76} C_VEL
LIN {X 0,Y 264.79,Z 956.392,A -85,B 0,C 180,E1 -18072.844,E2 -18072.844} C_VEL
LIN {X 0,Y 263.778,Z 961.265,A -85,B 0,C 180,E1 -18074.545,E2 -18074.545} C_VEL
LIN {X 0,Y 262.709,Z 966.64,A -85,B 0,C 180,E1 -18076.854,E2 -18076.854} C_VEL
LIN {X 0,Y 262.145,Z 970.926,A -85,B 0,C 180,E1 -18079.181,E2 -18079.181} C_VEL
LIN {X 0,Y 262.241,Z 977.574,A -85,B 0,C 180,E1 -18083.844,E2 -18083.844} C_VEL
LIN {X 0,Y 262.489,Z 979.293,A -85,B 0,C 180,E1 -18085.391,E2 -18085.391} C_VEL
LIN {X 0,Y 262.669,Z 980.565,A -85,B 0,C 180,E1 -18086.93,E2 -18086.93} C_VEL
LIN {X 0,Y 262.83,Z 981.398,A -85,B 0,C 180,E1 -18088.465,E2 -18088.465} C_VEL
LIN {X 0,Y 262.986,Z 981.762,A -85,B 0,C 180,E1 -18089.998,E2 -18089.998} C_VEL
LIN {X 0,Y 262.797,Z 981.66,A -85,B 0,C 180,E1 -18091.53,E2 -18091.53} C_VEL
LIN {X 0,Y 262.606,Z 981.146,A -85,B 0,C 180,E1 -18093.066,E2 -18093.066} C_VEL
LIN {X 0,Y 262.412,Z 980.215,A -85,B 0,C 180,E1 -18094.606,E2 -18094.606} C_VEL
LIN {X 0,Y 262.081,Z 977.698,A -85,B 0,C 180,E1 -18097.162,E2 -18097.162} C_VEL
LIN {X 0,Y 262.028,Z 973.433,A -85,B 0,C 180,E1 -18100.038,E2 -18100.038} C_VEL
LIN {X 0,Y 262.427,Z 968.814,A -85,B 0,C 180,E1 -18102.369,E2 -18102.369} C_VEL
LIN {X 0,Y 263.502,Z 961.96,A -85,B 0,C 180,E1 -18105.07,E2 -18105.07} C_VEL
LIN {X 0,Y 264.656,Z 955.632,A -85,B 0,C 180,E1 -18107.062,E2 -18107.062} C_VEL
LIN {X 0,Y 266.484,Z 947.143,A -85,B 0,C 180,E1 -18109.246,E2 -18109.246} C_VEL
LIN {X 0,Y 268.497,Z 938.229,A -85,B 0,C 180,E1 -18111.092,E2 -18111.092} C_VEL
LIN {X 0,Y 270.89,Z 927.344,A -85,B 0,C 180,E1 -18112.9,E2 -18112.9} C_VEL
LIN {X 0,Y 273.107,Z 916.599,A -85,B 0,C 180,E1 -18114.311,E2 -18114.311} C_VEL
LIN {X 0,Y 275.257,Z 904.69,A -85,B 0,C 180,E1 -18115.52,E2 -18115.52} C_VEL
LIN {X 0,Y 277.218,Z 891.124,A -85,B 0,C 180,E1 -18116.538,E2 -18116.538} C_VEL
LIN {X 0,Y 278.476,Z 878.386,A -85,B 0,C 180,E1 -18117.205,E2 -18117.205} C_VEL
LIN {X 0,Y 279.273,Z 861.967,A -85,B 0,C 180,E1 -18117.721,E2 -18117.721} C_VEL
LIN {X 0,Y 280.103,Z 835.254,A -85,B 0,C 180,E1 -18118.436,E2 -18118.436} C_VEL
LIN {X 0,Y 277.905,Z 807.31,A -85,B 0,C 180,E1 -18119.578,E2 -18119.578} C_VEL
LIN {X 0,Y 275.237,Z 783.505,A -85,B 0,C 180,E1 -18120.692,E2 -18120.692} C_VEL
LIN {X 0,Y 271.861,Z 761.699,A -85,B 0,C 180,E1 -18121.917,E2 -18121.917} C_VEL
LIN {X 0,Y 272.461,Z 757.969,A -85,B 0,C 180,E1 -18122.795,E2 -18122.795} C_VEL
LIN {X 0,Y 270.755,Z 748.458,A -85,B 0,C 180,E1 -18125.621,E2 -18125.621} C_VEL
LIN {X 0,Y 268.435,Z 738.198,A -85,B 0,C 180,E1 -18128.925,E2 -18128.925} C_VEL
LIN {X 0,Y 265.836,Z 728.836,A -85,B 0,C 180,E1 -18132.248,E2 -18132.248} C_VEL
LIN {X 0,Y 263.15,Z 719.821,A -85,B 0,C 180,E1 -18135.822,E2 -18135.822} C_VEL
LIN {X 0,Y 263.113,Z 719.694,A -85,B 0,C 180,E1 -18140.129,E2 -18140.129} C_VEL
LIN {X 0,Y 263.178,Z 719.683,A -85,B 0,C 180,E1 -18144.021,E2 -18144.021} C_VEL
LIN {X 0,Y 263.124,Z 719.71,A -85,B 0,C 180,E1 -18147.711,E2 -18147.711} C_VEL
LIN {X 0,Y 263.191,Z 719.695,A -85,B 0,C 180,E1 -18151.782,E2 -18151.782} C_VEL
LIN {X 0,Y 263.216,Z 719.691,A -85,B 0,C 180,E1 -18155.199,E2 -18155.199} C_VEL
LIN {X 0,Y 263.253,Z 719.688,A -85,B 0,C 180,E1 -18159.693,E2 -18159.693} C_VEL
LIN {X 0,Y 263.34,Z 719.682,A -85,B 0,C 180,E1 -18164.522,E2 -18164.522} C_VEL
LIN {X 0,Y 263.343,Z 719.682,A -85,B 0,C 180,E1 -18169.233,E2 -18169.233} C_VEL
LIN {X 0,Y 263.546,Z 719.649,A -85,B 0,C 180,E1 -18172.338,E2 -18172.338} C_VEL
LIN {X 0,Y 263.74,Z 719.631,A -85,B 0,C 180,E1 -18178.473,E2 -18178.473} C_VEL
LIN {X 0,Y 263.74,Z 719.628,A -85,B 0,C 180,E1 -18181.527,E2 -18181.527} C_VEL
LIN {X 0,Y 263.561,Z 719.65,A -85,B 0,C 180,E1 -18187.662,E2 -18187.662} C_VEL
LIN {X 0,Y 263.363,Z 719.681,A -85,B 0,C 180,E1 -18190.766,E2 -18190.766} C_VEL
LIN {X 0,Y 263.34,Z 719.675,A -85,B 0,C 180,E1 -18195.479,E2 -18195.479} C_VEL
LIN {X 0,Y 263.252,Z 719.692,A -85,B 0,C 180,E1 -18200.308,E2 -18200.308} C_VEL
LIN {X 0,Y 263.184,Z 719.692,A -85,B 0,C 180,E1 -18205.294,E2 -18205.294} C_VEL
LIN {X 0,Y 263.157,Z 719.688,A -85,B 0,C 180,E1 -18208.733,E2 -18208.733} C_VEL
LIN {X 0,Y 263.148,Z 719.889,A -85,B 0,C 180,E1 -18212.143,E2 -18212.143} C_VEL
LIN {X 0,Y 263.327,Z 720.768,A -85,B 0,C 180,E1 -18212.432,E2 -18212.432} C_VEL
LIN {X 0,Y 264.782,Z 723.475,A -85,B 0,C 180,E1 -18212.795,E2 -18212.795} C_VEL
LIN {X 0,Y 265.885,Z 725.072,A -85,B 0,C 180,E1 -18213.037,E2 -18213.037} C_VEL
LIN {X 0,Y 272.397,Z 735.988,A -85,B 0,C 180,E1 -18214.44,E2 -18214.44} C_VEL
LIN {X 0,Y 278.989,Z 748.435,A -85,B 0,C 180,E1 -18215.798,E2 -18215.798} C_VEL
LIN {X 0,Y 282.649,Z 756.224,A -85,B 0,C 180,E1 -18216.543,E2 -18216.543} C_VEL
LIN {X 0,Y 281.549,Z 798.344,A -85,B 0,C 180,E1 -18217.712,E2 -18217.712} C_VEL
LIN {X 0,Y 281.263,Z 811.903,A -85,B 0,C 180,E1 -18218.234,E2 -18218.234} C_VEL
